LIN {X 0,Y 239.536,Z 764.957,A -85,B 0,C 180,E1 -20171.852,E2 -20171.852} C_VEL
LIN {X 0,Y 237.019,Z 761.771,A -85,B 0,C 180,E1 -20173.722,E2 -20173.722} C_VEL
LIN {X 0,Y 235.633,Z 760.929,A -85,B 0,C 180,E1 -20174.686,E2 -20174.686} C_VEL
LIN {X 0,Y 233.822,Z 758.618,A -85,B 0,C 180,E1 -20176.248,E2 -20176.248} C_VEL
LIN {X 0,Y 232.796,Z 758.036,A -85,B 0,C 180,E1 -20177.061,E2 -20177.061} C_VEL
LIN {X 0,Y 230.567,Z 756.594,A -85,B 0,C 180,E1 -20179.103,E2 -20179.103} C_VEL
LIN {X 0,Y 229.613,Z 755.15,A -85,B 0,C 180,E1 -20180.375,E2 -20180.375} C_VEL
LIN {X 0,Y 230.024,Z 757.239,A -85,B 0,C 180,E1 -20185.325,E2 -20185.325} C_VEL
LIN {X 0,Y 230.532,Z 759.477,A -85,B 0,C 180,E1 -20189.195,E2 -20189.195} C_VEL
LIN {X 0,Y 231.145,Z 762.362,A -85,B 0,C 180,E1 -20193.181,E2 -20193.181} C_VEL
LIN {X 0,Y 232.117,Z 766.675,A -85,B 0,C 180,E1 -20198.073,E2 -20198.073} C_VEL
LIN {X 0,Y 232.844,Z 770.414,A -85,B 0,C 180,E1 -20201.608,E2 -20201.608} C_VEL
LIN {X 0,Y 233.498,Z 773.772,A -85,B 0,C 180,E1 -20204.335,E2 -20204.335} C_VEL
LIN {X 0,Y 235.393,Z 778.757,A -85,B 0,C 180,E1 -20205.95,E2 -20205.95} C_VEL
LIN {X 0,Y 237.78,Z 782.93,A -85,B 0,C 180,E1 -20207.6,E2 -20207.6} C_VEL
LIN {X 0,Y 239.967,Z 789.226,A -85,B 0,C 180,E1 -20209.271,E2 -20209.271} C_VEL
LIN {X 0,Y 241.097,Z 795.425,A -85,B 0,C 180,E1 -20210.543,E2 -20210.543} C_VEL
LIN {X 0,Y 241.775,Z 799.257,A -85,B 0,C 180,E1 -20211.301,E2 -20211.301} C_VEL
LIN {X 0,Y 241.913,Z 804.189,A -85,B 0,C 180,E1 -20212.077,E2 -20212.077} C_VEL
LIN {X 0,Y 241.291,Z 809.401,A -85,B 0,C 180,E1 -20212.744,E2 -20212.744} C_VEL
LIN {X 0,Y 238.925,Z 819.932,A -85,B 0,C 180,E1 -20214.02,E2 -20214.02} C_VEL
LIN {X 0,Y 238.088,Z 824.877,A -85,B 0,C 180,E1 -20214.79,E2 -20214.79} C_VEL
LIN {X 0,Y 238.001,Z 826.424,A -85,B 0,C 180,E1 -20215.084,E2 -20215.084} C_VEL
LIN {X 0,Y 237.022,Z 838.207,A -85,B 0,C 180,E1 -20217.458,E2 -20217.458} C_VEL
LIN {X 0,Y 234.947,Z 849.621,A -85,B 0,C 180,E1 -20219.926,E2 -20219.926} C_VEL
LIN {X 0,Y 231.947,Z 860.19,A -85,B 0,C 180,E1 -20222.479,E2 -20222.479} C_VEL
LIN {X 0,Y 229.183,Z 869.039,A -85,B 0,C 180,E1 -20225.061,E2 -20225.061} C_VEL
LIN {X 0,Y 226.722,Z 875.341,A -85,B 0,C 180,E1 -20227.202,E2 -20227.202} C_VEL
LIN {X 0,Y 223.981,Z 881.748,A -85,B 0,C 180,E1 -20229.808,E2 -20229.808} C_VEL
LIN {X 0,Y 221.954,Z 887.028,A -85,B 0,C 180,E1 -20232.493,E2 -20232.493} C_VEL
LIN {X 0,Y 220.653,Z 891.327,A -85,B 0,C 180,E1 -20235.238,E2 -20235.238} C_VEL
LIN {X 0,Y 219.689,Z 895.654,A -85,B 0,C 180,E1 -20238.933,E2 -20238.933} C_VEL
LIN {X 0,Y 219.717,Z 898.373,A -85,B 0,C 180,E1 -20242.649,E2 -20242.649} C_VEL
LIN {X 0,Y 219.985,Z 899.167,A -85,B 0,C 180,E1 -20244.5,E2 -20244.5} C_VEL
LIN {X 0,Y 220.278,Z 899.554,A -85,B 0,C 180,E1 -20246.341,E2 -20246.341} C_VEL
LIN {X 0,Y 220.658,Z 899.53,A -85,B 0,C 180,E1 -20248.175,E2 -20248.175} C_VEL
LIN {X 0,Y 221.137,Z 899.063,A -85,B 0,C 180,E1 -20250,E2 -20250} C_VEL
LIN {X 0,Y 220.915,Z 898.036,A -85,B 0,C 180,E1 -20251.823,E2 -20251.823} C_VEL
LIN {X 0,Y 220.65,Z 896.554,A -85,B 0,C 180,E1 -20253.652,E2 -20253.652} C_VEL
LIN {X 0,Y 220.44,Z 893.409,A -85,B 0,C 180,E1 -20256.407,E2 -20256.407} C_VEL
LIN {X 0,Y 220.219,Z 889.055,A -85,B 0,C 180,E1 -20259.182,E2 -20259.182} C_VEL
LIN {X 0,Y 220.533,Z 882.364,A -85,B 0,C 180,E1 -20262.422,E2 -20262.422} C_VEL
LIN {X 0,Y 221.328,Z 875.061,A -85,B 0,C 180,E1 -20265.187,E2 -20265.187} C_VEL
LIN {X 0,Y 222.405,Z 867.639,A -85,B 0,C 180,E1 -20267.47,E2 -20267.47} C_VEL
LIN {X 0,Y 223.753,Z 859.408,A -85,B 0,C 180,E1 -20269.56,E2 -20269.56} C_VEL
LIN {X 0,Y 223.898,Z 849.535,A -85,B 0,C 180,E1 -20271.643,E2 -20271.643} C_VEL
LIN {X 0,Y 223.822,Z 838.205,A -85,B 0,C 180,E1 -20273.6,E2 -20273.6} C_VEL
LIN {X 0,Y 223.429,Z 825.557,A -85,B 0,C 180,E1 -20275.376,E2 -20275.376} C_VEL
LIN {X 0,Y 222.909,Z 813.807,A -85,B 0,C 180,E1 -20276.684,E2 -20276.684} C_VEL
LIN {X 0,Y 222.051,Z 799.54,A -85,B 0,C 180,E1 -20277.884,E2 -20277.884} C_VEL
LIN {X 0,Y 221.631,Z 793.027,A -85,B 0,C 180,E1 -20278.33,E2 -20278.33} C_VEL
LIN {X 0,Y 223.268,Z 783.83,A -85,B 0,C 180,E1 -20283.426,E2 -20283.426} C_VEL
LIN {X 0,Y 225.052,Z 776.429,A -85,B 0,C 180,E1 -20287.514,E2 -20287.514} C_VEL
LIN {X 0,Y 225.493,Z 774.103,A -85,B 0,C 180,E1 -20288.814,E2 -20288.814} C_VEL
LIN {X 0,Y 225.149,Z 770.421,A -85,B 0,C 180,E1 -20290.959,E2 -20290.959} C_VEL
LIN {X 0,Y 223.734,Z 763.752,A -85,B 0,C 180,E1 -20295.027,E2 -20295.027} C_VEL
LIN {X 0,Y 222.198,Z 755.968,A -85,B 0,C 180,E1 -20300.027,E2 -20300.027} C_VEL
LIN {X 0,Y 220.923,Z 748.963,A -85,B 0,C 180,E1 -20304.789,E2 -20304.789} C_VEL
LIN {X 0,Y 220.869,Z 748.973,A -85,B 0,C 180,E1 -20309.395,E2 -20309.395} C_VEL
LIN {X 0,Y 220.896,Z 748.965,A -85,B 0,C 180,E1 -20313.55,E2 -20313.55} C_VEL
LIN {X 0,Y 220.867,Z 748.972,A -85,B 0,C 180,E1 -20317.552,E2 -20317.552} C_VEL
LIN {X 0,Y 220.986,Z 748.956,A -85,B 0,C 180,E1 -20322.571,E2 -20322.571} C_VEL
LIN {X 0,Y 221.014,Z 748.952,A -85,B 0,C 180,E1 -20327.139,E2 -20327.139} C_VEL
LIN {X 0,Y 221.207,Z 748.927,A -85,B 0,C 180,E1 -20330.86,E2 -20330.86} C_VEL
LIN {X 0,Y 221.261,Z 748.924,A -85,B 0,C 180,E1 -20332.701,E2 -20332.701} C_VEL
LIN {X 0,Y 221.509,Z 748.89,A -85,B 0,C 180,E1 -20338.182,E2 -20338.182} C_VEL
LIN {X 0,Y 221.51,Z 748.89,A -85,B 0,C 180,E1 -20341.818,E2 -20341.818} C_VEL
LIN {X 0,Y 221.243,Z 748.922,A -85,B 0,C 180,E1 -20347.3,E2 -20347.3} C_VEL
LIN {X 0,Y 221.064,Z 748.95,A -85,B 0,C 180,E1 -20350.997,E2 -20350.997} C_VEL
LIN {X 0,Y 220.992,Z 748.953,A -85,B 0,C 180,E1 -20356.632,E2 -20356.632} C_VEL
LIN {X 0,Y 220.876,Z 748.97,A -85,B 0,C 180,E1 -20360.488,E2 -20360.488} C_VEL
LIN {X 0,Y 220.8,Z 748.976,A -85,B 0,C 180,E1 -20364.443,E2 -20364.443} C_VEL
LIN {X 0,Y 220.801,Z 748.979,A -85,B 0,C 180,E1 -20368.519,E2 -20368.519} C_VEL
LIN {X 0,Y 220.813,Z 748.975,A -85,B 0,C 180,E1 -20372.757,E2 -20372.757} C_VEL
LIN {X 0,Y 220.797,Z 748.98,A -85,B 0,C 180,E1 -20377.274,E2 -20377.274} C_VEL
LIN {X 0,Y 220.747,Z 748.985,A -85,B 0,C 180,E1 -20381.958,E2 -20381.958} C_VEL
LIN {X 0,Y 220.753,Z 748.986,A -85,B 0,C 180,E1 -20385.541,E2 -20385.541} C_VEL
LIN {X 0,Y 220.781,Z 748.979,A -85,B 0,C 180,E1 -20390.458,E2 -20390.458} C_VEL
LIN {X 0,Y 220.826,Z 748.975,A -85,B 0,C 180,E1 -20392.793,E2 -20392.793} C_VEL
LIN {X 0,Y 220.812,Z 748.977,A -85,B 0,C 180,E1 -20397.243,E2 -20397.243} C_VEL
LIN {X 0,Y 220.793,Z 748.978,A -85,B 0,C 180,E1 -20401.48,E2 -20401.48} C_VEL
LIN {X 0,Y 220.806,Z 748.978,A -85,B 0,C 180,E1 -20405.558,E2 -20405.558} C_VEL
LIN {X 0,Y 220.876,Z 748.967,A -85,B 0,C 180,E1 -20409.512,E2 -20409.512} C_VEL
LIN {X 0,Y 220.981,Z 748.957,A -85,B 0,C 180,E1 -20413.368,E2 -20413.368} C_VEL
LIN {X 0,Y 221.064,Z 748.949,A -85,B 0,C 180,E1 -20419.004,E2 -20419.004} C_VEL
LIN {X 0,Y 221.24,Z 748.926,A -85,B 0,C 180,E1 -20422.7,E2 -20422.7} C_VEL
LIN {X 0,Y 221.471,Z 748.895,A -85,B 0,C 180,E1 -20428.182,E2 -20428.182} C_VEL
LIN {X 0,Y 221.471,Z 748.895,A -85,B 0,C 180,E1 -20431.819,E2 -20431.819} C_VEL
LIN {X 0,Y 221.241,Z 748.927,A -85,B 0,C 180,E1 -20437.3,E2 -20437.3} C_VEL
LIN {X 0,Y 221.069,Z 748.946,A -85,B 0,C 180,E1 -20440.997,E2 -20440.997} C_VEL
LIN {X 0,Y 221.02,Z 748.951,A -85,B 0,C 180,E1 -20446.63,E2 -20446.63} C_VEL
LIN {X 0,Y 220.89,Z 748.966,A -85,B 0,C 180,E1 -20450.487,E2 -20450.487} C_VEL
LIN {X 0,Y 220.85,Z 748.973,A -85,B 0,C 180,E1 -20454.437,E2 -20454.437} C_VEL
LIN {X 0,Y 220.807,Z 748.979,A -85,B 0,C 180,E1 -20458.518,E2 -20458.518} C_VEL
LIN {X 0,Y 220.815,Z 748.978,A -85,B 0,C 180,E1 -20462.757,E2 -20462.757} C_VEL
LIN {X 0,Y 220.872,Z 748.986,A -85,B 0,C 180,E1 -20465.851,E2 -20465.851} C_VEL
LIN {X 0,Y 224.644,Z 761.399,A -85,B 0,C 180,E1 -20467.576,E2 -20467.576} C_VEL
LIN {X 0,Y 228.039,Z 773.686,A -85,B 0,C 180,E1 -20469.602,E2 -20469.602} C_VEL
LIN {X 0,Y 228.898,Z 778.294,A -85,B 0,C 180,E1 -20470.437,E2 -20470.437} C_VEL
LIN {X 0,Y 227.328,Z 790.026,A -85,B 0,C 180,E1 -20472.609,E2 -20472.609} C_VEL
LIN {X 0,Y 225.869,Z 799.76,A -85,B 0,C 180,E1 -20474.822,E2 -20474.822} C_VEL
LIN {X 0,Y 224.622,Z 808.015,A -85,B 0,C 180,E1 -20477.116,E2 -20477.116} C_VEL
LIN {X 0,Y 223.342,Z 816.261,A -85,B 0,C 180,E1 -20479.924,E2 -20479.924} C_VEL
LIN {X 0,Y 222.478,Z 822.628,A -85,B 0,C 180,E1 -20482.611,E2 -20482.611} C_VEL
LIN {X 0,Y 221.94,Z 827.949,A -85,B 0,C 180,E1 -20485.42,E2 -20485.42} C_VEL
LIN {X 0,Y 221.554,Z 832.917,A -85,B 0,C 180,E1 -20488.924,E2 -20488.924} C_VEL
LIN {X 0,Y 221.741,Z 836.407,A -85,B 0,C 180,E1 -20492.556,E2 -20492.556} C_VEL
LIN {X 0,Y 222.586,Z 838.266,A -85,B 0,C 180,E1 -20496.3,E2 -20496.3} C_VEL
LIN {X 0,Y 223.975,Z 838.52,A -85,B 0,C 180,E1 -20499.808,E2 -20499.808} C_VEL
LIN {X 0,Y 225.01,Z 837.966,A -85,B 0,C 180,E1 -20501.799,E2 -20501.799} C_VEL
LIN {X 0,Y 226.495,Z 836.725,A -85,B 0,C 180,E1 -20504.137,E2 -20504.137} C_VEL
LIN {X 0,Y 229.235,Z 833.462,A -85,B 0,C 180,E1 -20507.607,E2 -20507.607} C_VEL
LIN {X 0,Y 232.035,Z 829.448,A -85,B 0,C 180,E1 -20510.41,E2 -20510.41} C_VEL
LIN {X 0,Y 235.262,Z 824.148,A -85,B 0,C 180,E1 -20513.137,E2 -20513.137} C_VEL
LIN {X 0,Y 238.765,Z 817.443,A -85,B 0,C 180,E1 -20515.778,E2 -20515.778} C_VEL
LIN {X 0,Y 242.054,Z 810.487,A -85,B 0,C 180,E1 -20517.92,E2 -20517.92} C_VEL
LIN {X 0,Y 245.491,Z 802.175,A -85,B 0,C 180,E1 -20520,E2 -20520} C_VEL
LIN {X 0,Y 245.181,Z 797.388,A -85,B 0,C 180,E1 -20521.642,E2 -20521.642} C_VEL
LIN {X 0,Y 244.015,Z 789.753,A -85,B 0,C 180,E1 -20524.236,E2 -20524.236} C_VEL
LIN {X 0,Y 242.382,Z 784.469,A -85,B 0,C 180,E1 -20526.227,E2 -20526.227} C_VEL
LIN {X 0,Y 238.461,Z 774.826,A -85,B 0,C 180,E1 -20530.185,E2 -20530.185} C_VEL
LIN {X 0,Y 236.378,Z 771.366,A -85,B 0,C 180,E1 -20532.012,E2 -20532.012} C_VEL
LIN {X 0,Y 234.167,Z 768.376,A -85,B 0,C 180,E1 -20533.892,E2 -20533.892} C_VEL
LIN {X 0,Y 229.777,Z 764.406,A -85,B 0,C 180,E1 -20537.81,E2 -20537.81} C_VEL
LIN {X 0,Y 227.615,Z 762.171,A -85,B 0,C 180,E1 -20540.373,E2 -20540.373} C_VEL
LIN {X 0,Y 224.085,Z 761.37,A -85,B 0,C 180,E1 -20546.045,E2 -20546.045} C_VEL
LIN {X 0,Y 223.685,Z 761.148,A -85,B 0,C 180,E1 -20548.118,E2 -20548.118} C_VEL
LIN {X 0,Y 224.259,Z 763.902,A -85,B 0,C 180,E1 -20552.204,E2 -20552.204} C_VEL
LIN {X 0,Y 225.112,Z 767.836,A -85,B 0,C 180,E1 -20556.801,E2 -20556.801} C_VEL
LIN {X 0,Y 228.683,Z 776.557,A -85,B 0,C 180,E1 -20561.863,E2 -20561.863} C_VEL
LIN {X 0,Y 230.667,Z 779.851,A -85,B 0,C 180,E1 -20563.67,E2 -20563.67} C_VEL
LIN {X 0,Y 232.193,Z 784.445,A -85,B 0,C 180,E1 -20565.254,E2 -20565.254} C_VEL
LIN {X 0,Y 234.205,Z 788.172,A -85,B 0,C 180,E1 -20566.81,E2 -20566.81} C_VEL
LIN {X 0,Y 235.872,Z 793.983,A -85,B 0,C 180,E1 -20568.434,E2 -20568.434} C_VEL
LIN {X 0,Y 237.128,Z 803.079,A -85,B 0,C 180,E1 -20570.407,E2 -20570.407} C_VEL
LIN {X 0,Y 238.077,Z 816.236,A -85,B 0,C 180,E1 -20573.062,E2 -20573.062} C_VEL
LIN {X 0,Y 238.001,Z 826.424,A -85,B 0,C 180,E1 -20575.084,E2 -20575.084} C_VEL
LIN {X 0,Y 237.26,Z 831.186,A -85,B 0,C 180,E1 -20575.915,E2 -20575.915} C_VEL
LIN {X 0,Y 235.527,Z 836.054,A -85,B 0,C 180,E1 -20576.636,E2 -20576.636} C_VEL
LIN {X 0,Y 230.95,Z 845.512,A -85,B 0,C 180,E1 -20578.063,E2 -20578.063} C_VEL
LIN {X 0,Y 229.043,Z 849.964,A -85,B 0,C 180,E1 -20578.936,E2 -20578.936} C_VEL
LIN {X 0,Y 228.592,Z 851.381,A -85,B 0,C 180,E1 -20579.268,E2 -20579.268} C_VEL
LIN {X 0,Y 225.114,Z 862.094,A -85,B 0,C 180,E1 -20582.076,E2 -20582.076} C_VEL
LIN {X 0,Y 221.765,Z 871.694,A -85,B 0,C 180,E1 -20585.171,E2 -20585.171} C_VEL
LIN {X 0,Y 218.161,Z 879.44,A -85,B 0,C 180,E1 -20588.255,E2 -20588.255} C_VEL
LIN {X 0,Y 215.692,Z 884.912,A -85,B 0,C 180,E1 -20590.984,E2 -20590.984} C_VEL
LIN {X 0,Y 213.728,Z 890.678,A -85,B 0,C 180,E1 -20594.748,E2 -20594.748} C_VEL
LIN {X 0,Y 212.66,Z 894.779,A -85,B 0,C 180,E1 -20598.563,E2 -20598.563} C_VEL
LIN {X 0,Y 212.673,Z 897.416,A -85,B 0,C 180,E1 -20602.472,E2 -20602.472} C_VEL
LIN {X 0,Y 212.925,Z 898.116,A -85,B 0,C 180,E1 -20604.317,E2 -20604.317} C_VEL
LIN {X 0,Y 213.224,Z 898.43,A -85,B 0,C 180,E1 -20606.22,E2 -20606.22} C_VEL
LIN {X 0,Y 213.649,Z 898.324,A -85,B 0,C 180,E1 -20608.115,E2 -20608.115} C_VEL
LIN {X 0,Y 214.155,Z 897.813,A -85,B 0,C 180,E1 -20610,E2 -20610} C_VEL
LIN {X 0,Y 213.897,Z 896.725,A -85,B 0,C 180,E1 -20611.883,E2 -20611.883} C_VEL
LIN {X 0,Y 213.551,Z 894.183,A -85,B 0,C 180,E1 -20614.719,E2 -20614.719} C_VEL
LIN {X 0,Y 213.289,Z 890.503,A -85,B 0,C 180,E1 -20617.574,E2 -20617.574} C_VEL
LIN {X 0,Y 213.233,Z 885.6,A -85,B 0,C 180,E1 -20620.444,E2 -20620.444} C_VEL
LIN {X 0,Y 213.686,Z 879.386,A -85,B 0,C 180,E1 -20623.31,E2 -20623.31} C_VEL
LIN {X 0,Y 214.678,Z 871.586,A -85,B 0,C 180,E1 -20626.157,E2 -20626.157} C_VEL
LIN {X 0,Y 216.168,Z 861.923,A -85,B 0,C 180,E1 -20628.973,E2 -20628.973} C_VEL
LIN {X 0,Y 216.716,Z 856.865,A -85,B 0,C 180,E1 -20630.204,E2 -20630.204} C_VEL
LIN {X 0,Y 216.786,Z 846.465,A -85,B 0,C 180,E1 -20632.391,E2 -20632.391} C_VEL
LIN {X 0,Y 216.675,Z 834.784,A -85,B 0,C 180,E1 -20634.412,E2 -20634.412} C_VEL
LIN {X 0,Y 216.312,Z 822.268,A -85,B 0,C 180,E1 -20636.145,E2 -20636.145} C_VEL
LIN {X 0,Y 215.674,Z 808.554,A -85,B 0,C 180,E1 -20637.634,E2 -20637.634} C_VEL
LIN {X 0,Y 214.841,Z 794.999,A -85,B 0,C 180,E1 -20638.711,E2 -20638.711} C_VEL
LIN {X 0,Y 214.664,Z 792.094,A -85,B 0,C 180,E1 -20638.898,E2 -20638.898} C_VEL
LIN {X 0,Y 216.195,Z 783.992,A -85,B 0,C 180,E1 -20643.548,E2 -20643.548} C_VEL
LIN {X 0,Y 218.355,Z 775.24,A -85,B 0,C 180,E1 -20648.578,E2 -20648.578} C_VEL
LIN {X 0,Y 218.388,Z 772.741,A -85,B 0,C 180,E1 -20650.063,E2 -20650.063} C_VEL
LIN {X 0,Y 217.183,Z 766.986,A -85,B 0,C 180,E1 -20653.626,E2 -20653.626} C_VEL
LIN {X 0,Y 215.615,Z 759.392,A -85,B 0,C 180,E1 -20658.563,E2 -20658.563} C_VEL
LIN {X 0,Y 214.486,Z 753.23,A -85,B 0,C 180,E1 -20662.79,E2 -20662.79} C_VEL
LIN {X 0,Y 213.855,Z 749.844,A -85,B 0,C 180,E1 -20665.244,E2 -20665.244} C_VEL
LIN {X 0,Y 213.782,Z 749.853,A -85,B 0,C 180,E1 -20670.454,E2 -20670.454} C_VEL
LIN {X 0,Y 213.8,Z 749.85,A -85,B 0,C 180,E1 -20674.702,E2 -20674.702} C_VEL
LIN {X 0,Y 213.805,Z 749.85,A -85,B 0,C 180,E1 -20678.803,E2 -20678.803} C_VEL
LIN {X 0,Y 213.945,Z 749.832,A -85,B 0,C 180,E1 -20682.804,E2 -20682.804} C_VEL
LIN {X 0,Y 213.955,Z 749.833,A -85,B 0,C 180,E1 -20686.707,E2 -20686.707} C_VEL
LIN {X 0,Y 214.144,Z 749.808,A -85,B 0,C 180,E1 -20690.555,E2 -20690.555} C_VEL
LIN {X 0,Y 214.096,Z 749.817,A -85,B 0,C 180,E1 -20694.349,E2 -20694.349} C_VEL
LIN {X 0,Y 214.442,Z 749.77,A -85,B 0,C 180,E1 -20698.122,E2 -20698.122} C_VEL
LIN {X 0,Y 214.544,Z 749.756,A -85,B 0,C 180,E1 -20700,E2 -20700} C_VEL
LIN {X 0,Y 214.443,Z 749.77,A -85,B 0,C 180,E1 -20701.878,E2 -20701.878} C_VEL
LIN {X 0,Y 214.184,Z 749.8,A -85,B 0,C 180,E1 -20707.542,E2 -20707.542} C_VEL
LIN {X 0,Y 213.995,Z 749.828,A -85,B 0,C 180,E1 -20711.365,E2 -20711.365} C_VEL
LIN {X 0,Y 213.91,Z 749.837,A -85,B 0,C 180,E1 -20715.239,E2 -20715.239} C_VEL
LIN {X 0,Y 213.82,Z 749.851,A -85,B 0,C 180,E1 -20719.189,E2 -20719.189} C_VEL
LIN {X 0,Y 213.784,Z 749.855,A -85,B 0,C 180,E1 -20723.235,E2 -20723.235} C_VEL
LIN {X 0,Y 213.786,Z 749.855,A -85,B 0,C 180,E1 -20727.427,E2 -20727.427} C_VEL
LIN {X 0,Y 213.76,Z 749.857,A -85,B 0,C 180,E1 -20731.739,E2 -20731.739} C_VEL
LIN {X 0,Y 213.742,Z 749.859,A -85,B 0,C 180,E1 -20736.289,E2 -20736.289} C_VEL
LIN {X 0,Y 213.697,Z 749.863,A -85,B 0,C 180,E1 -20741.129,E2 -20741.129} C_VEL
LIN {X 0,Y 213.702,Z 749.863,A -85,B 0,C 180,E1 -20743.68,E2 -20743.68} C_VEL
LIN {X 0,Y 213.702,Z 749.865,A -85,B 0,C 180,E1 -20746.346,E2 -20746.346} C_VEL
LIN {X 0,Y 213.702,Z 749.859,A -85,B 0,C 180,E1 -20751.329,E2 -20751.329} C_VEL
LIN {X 0,Y 213.755,Z 749.859,A -85,B 0,C 180,E1 -20756.018,E2 -20756.018} C_VEL
LIN {X 0,Y 213.746,Z 749.858,A -85,B 0,C 180,E1 -20760.449,E2 -20760.449} C_VEL
LIN {X 0,Y 213.742,Z 749.86,A -85,B 0,C 180,E1 -20764.694,E2 -20764.694} C_VEL
LIN {X 0,Y 213.795,Z 749.852,A -85,B 0,C 180,E1 -20768.802,E2 -20768.802} C_VEL
LIN {X 0,Y 213.895,Z 749.842,A -85,B 0,C 180,E1 -20772.8,E2 -20772.8} C_VEL
LIN {X 0,Y 213.937,Z 749.834,A -85,B 0,C 180,E1 -20776.706,E2 -20776.706} C_VEL
LIN {X 0,Y 214.136,Z 749.81,A -85,B 0,C 180,E1 -20780.555,E2 -20780.555} C_VEL
LIN {X 0,Y 214.076,Z 749.816,A -85,B 0,C 180,E1 -20784.348,E2 -20784.348} C_VEL
LIN {X 0,Y 214.407,Z 749.775,A -85,B 0,C 180,E1 -20788.122,E2 -20788.122} C_VEL
LIN {X 0,Y 214.515,Z 749.762,A -85,B 0,C 180,E1 -20790,E2 -20790} C_VEL
LIN {X 0,Y 214.408,Z 749.775,A -85,B 0,C 180,E1 -20791.879,E2 -20791.879} C_VEL
LIN {X 0,Y 214.183,Z 749.806,A -85,B 0,C 180,E1 -20797.542,E2 -20797.542} C_VEL
LIN {X 0,Y 214.001,Z 749.828,A -85,B 0,C 180,E1 -20801.365,E2 -20801.365} C_VEL
LIN {X 0,Y 213.936,Z 749.834,A -85,B 0,C 180,E1 -20805.237,E2 -20805.237} C_VEL
LIN {X 0,Y 213.84,Z 749.847,A -85,B 0,C 180,E1 -20809.188,E2 -20809.188} C_VEL
LIN {X 0,Y 213.806,Z 749.851,A -85,B 0,C 180,E1 -20813.232,E2 -20813.232} C_VEL
LIN {X 0,Y 213.79,Z 749.854,A -85,B 0,C 180,E1 -20817.428,E2 -20817.428} C_VEL
LIN {X 0,Y 213.761,Z 749.859,A -85,B 0,C 180,E1 -20821.739,E2 -20821.739} C_VEL
LIN {X 0,Y 213.794,Z 749.853,A -85,B 0,C 180,E1 -20825.294,E2 -20825.294} C_VEL
LIN {X 0,Y 217.876,Z 763.131,A -85,B 0,C 180,E1 -20827.216,E2 -20827.216} C_VEL
LIN {X 0,Y 220.84,Z 774.127,A -85,B 0,C 180,E1 -20829.093,E2 -20829.093} C_VEL
LIN {X 0,Y 221.943,Z 778.391,A -85,B 0,C 180,E1 -20829.91,E2 -20829.91} C_VEL
LIN {X 0,Y 220.775,Z 788.422,A -85,B 0,C 180,E1 -20831.762,E2 -20831.762} C_VEL
LIN {X 0,Y 219.117,Z 798.981,A -85,B 0,C 180,E1 -20834.138,E2 -20834.138} C_VEL
LIN {X 0,Y 217.708,Z 808.187,A -85,B 0,C 180,E1 -20836.686,E2 -20836.686} C_VEL
LIN {X 0,Y 216.409,Z 816.36,A -85,B 0,C 180,E1 -20839.495,E2 -20839.495} C_VEL
LIN {X 0,Y 215.312,Z 824.119,A -85,B 0,C 180,E1 -20842.853,E2 -20842.853} C_VEL
LIN {X 0,Y 214.73,Z 830.013,A -85,B 0,C 180,E1 -20846.192,E2 -20846.192} C_VEL
LIN {X 0,Y 214.471,Z 834.375,A -85,B 0,C 180,E1 -20849.487,E2 -20849.487} C_VEL
LIN {X 0,Y 214.739,Z 837.379,A -85,B 0,C 180,E1 -20852.729,E2 -20852.729} C_VEL
LIN {X 0,Y 215.445,Z 839.173,A -85,B 0,C 180,E1 -20855.978,E2 -20855.978} C_VEL
LIN {X 0,Y 216.991,Z 839.729,A -85,B 0,C 180,E1 -20859.93,E2 -20859.93} C_VEL
LIN {X 0,Y 219.341,Z 838.449,A -85,B 0,C 180,E1 -20863.997,E2 -20863.997} C_VEL
LIN {X 0,Y 221.803,Z 836.025,A -85,B 0,C 180,E1 -20867.185,E2 -20867.185} C_VEL
LIN {X 0,Y 224.581,Z 832.601,A -85,B 0,C 180,E1 -20870.089,E2 -20870.089} C_VEL
LIN {X 0,Y 227.856,Z 827.892,A -85,B 0,C 180,E1 -20872.913,E2 -20872.913} C_VEL
LIN {X 0,Y 231.435,Z 821.837,A -85,B 0,C 180,E1 -20875.647,E2 -20875.647} C_VEL
LIN {X 0,Y 235.499,Z 814.219,A -85,B 0,C 180,E1 -20878.29,E2 -20878.29} C_VEL
LIN {X 0,Y 239.404,Z 805.721,A -85,B 0,C 180,E1 -20880.588,E2 -20880.588} C_VEL
LIN {X 0,Y 239.801,Z 804.702,A -85,B 0,C 180,E1 -20880.839,E2 -20880.839} C_VEL
LIN {X 0,Y 239.135,Z 795.516,A -85,B 0,C 180,E1 -20884.213,E2 -20884.213} C_VEL
LIN {X 0,Y 238.04,Z 790.733,A -85,B 0,C 180,E1 -20886.083,E2 -20886.083} C_VEL
LIN {X 0,Y 234.694,Z 780.967,A -85,B 0,C 180,E1 -20890.351,E2 -20890.351} C_VEL
LIN {X 0,Y 232.945,Z 777.567,A -85,B 0,C 180,E1 -20892.192,E2 -20892.192} C_VEL
LIN {X 0,Y 231.028,Z 774.762,A -85,B 0,C 180,E1 -20894.085,E2 -20894.085} C_VEL
LIN {X 0,Y 227.118,Z 770.93,A -85,B 0,C 180,E1 -20898.025,E2 -20898.025} C_VEL
LIN {X 0,Y 225.244,Z 768.855,A -85,B 0,C 180,E1 -20900.6,E2 -20900.6} C_VEL
LIN {X 0,Y 222.86,Z 768.528,A -85,B 0,C 180,E1 -20904.202,E2 -20904.202} C_VEL
LIN {X 0,Y 221.879,Z 768.004,A -85,B 0,C 180,E1 -20907.969,E2 -20907.969} C_VEL
LIN {X 0,Y 221.79,Z 771.249,A -85,B 0,C 180,E1 -20912.999,E2 -20912.999} C_VEL
LIN {X 0,Y 223.048,Z 774.544,A -85,B 0,C 180,E1 -20916.471,E2 -20916.471} C_VEL
LIN {X 0,Y 227.449,Z 785.277,A -85,B 0,C 180,E1 -20922.827,E2 -20922.827} C_VEL
LIN {X 0,Y 229.085,Z 790.743,A -85,B 0,C 180,E1 -20924.879,E2 -20924.879} C_VEL
LIN {X 0,Y 230.442,Z 793.382,A -85,B 0,C 180,E1 -20926.03,E2 -20926.03} C_VEL
LIN {X 0,Y 231.488,Z 797.369,A -85,B 0,C 180,E1 -20927.262,E2 -20927.262} C_VEL
LIN {X 0,Y 232.472,Z 807.335,A -85,B 0,C 180,E1 -20929.584,E2 -20929.584} C_VEL
LIN {X 0,Y 232.808,Z 820.657,A -85,B 0,C 180,E1 -20932.471,E2 -20932.471} C_VEL
LIN {X 0,Y 232.104,Z 831.966,A -85,B 0,C 180,E1 -20934.878,E2 -20934.878} C_VEL
LIN {X 0,Y 230.559,Z 842.773,A -85,B 0,C 180,E1 -20937.244,E2 -20937.244} C_VEL
LIN {X 0,Y 228.592,Z 851.381,A -85,B 0,C 180,E1 -20939.268,E2 -20939.268} C_VEL
LIN {X 0,Y 226.806,Z 855.608,A -85,B 0,C 180,E1 -20940.226,E2 -20940.226} C_VEL
LIN {X 0,Y 222.111,Z 862.268,A -85,B 0,C 180,E1 -20941.674,E2 -20941.674} C_VEL
LIN {X 0,Y 218.121,Z 867.224,A -85,B 0,C 180,E1 -20942.914,E2 -20942.914} C_VEL
LIN {X 0,Y 215.772,Z 870.701,A -85,B 0,C 180,E1 -20944.012,E2 -20944.012} C_VEL
LIN {X 0,Y 215.23,Z 871.789,A -85,B 0,C 180,E1 -20944.42,E2 -20944.42} C_VEL
LIN {X 0,Y 211.542,Z 879.206,A -85,B 0,C 180,E1 -20947.538,E2 -20947.538} C_VEL
LIN {X 0,Y 208.958,Z 884.455,A -85,B 0,C 180,E1 -20950.346,E2 -20950.346} C_VEL
LIN {X 0,Y 207.254,Z 888.754,A -85,B 0,C 180,E1 -20953.247,E2 -20953.247} C_VEL
LIN {X 0,Y 206.077,Z 892.144,A -85,B 0,C 180,E1 -20956.188,E2 -20956.188} C_VEL
LIN {X 0,Y 205.481,Z 895.334,A -85,B 0,C 180,E1 -20960.153,E2 -20960.153} C_VEL
LIN {X 0,Y 205.618,Z 896.491,A -85,B 0,C 180,E1 -20962.402,E2 -20962.402} C_VEL
LIN {X 0,Y 205.867,Z 897.031,A -85,B 0,C 180,E1 -20964.121,E2 -20964.121} C_VEL
LIN {X 0,Y 206.634,Z 897.094,A -85,B 0,C 180,E1 -20968.051,E2 -20968.051} C_VEL
LIN {X 0,Y 207.165,Z 896.532,A -85,B 0,C 180,E1 -20970,E2 -20970} C_VEL
LIN {X 0,Y 206.878,Z 895.374,A -85,B 0,C 180,E1 -20971.947,E2 -20971.947} C_VEL
LIN {X 0,Y 206.543,Z 892.724,A -85,B 0,C 180,E1 -20974.88,E2 -20974.88} C_VEL
LIN {X 0,Y 206.251,Z 888.909,A -85,B 0,C 180,E1 -20977.834,E2 -20977.834} C_VEL
LIN {X 0,Y 206.24,Z 883.853,A -85,B 0,C 180,E1 -20980.802,E2 -20980.802} C_VEL
LIN {X 0,Y 206.784,Z 877.45,A -85,B 0,C 180,E1 -20983.763,E2 -20983.763} C_VEL
LIN {X 0,Y 207.853,Z 869.469,A -85,B 0,C 180,E1 -20986.703,E2 -20986.703} C_VEL
LIN {X 0,Y 209.132,Z 861.336,A -85,B 0,C 180,E1 -20989.126,E2 -20989.126} C_VEL
LIN {X 0,Y 209.624,Z 856.536,A -85,B 0,C 180,E1 -20990.357,E2 -20990.357} C_VEL
LIN {X 0,Y 209.738,Z 846.049,A -85,B 0,C 180,E1 -20992.665,E2 -20992.665} C_VEL
LIN {X 0,Y 209.641,Z 834.841,A -85,B 0,C 180,E1 -20994.699,E2 -20994.699} C_VEL
LIN {X 0,Y 209.356,Z 822.205,A -85,B 0,C 180,E1 -20996.545,E2 -20996.545} C_VEL
LIN {X 0,Y 208.74,Z 808.282,A -85,B 0,C 180,E1 -20998.123,E2 -20998.123} C_VEL
LIN {X 0,Y 207.906,Z 794.49,A -85,B 0,C 180,E1 -20999.275,E2 -20999.275} C_VEL
LIN {X 0,Y 207.768,Z 791.111,A -85,B 0,C 180,E1 -20999.527,E2 -20999.527} C_VEL
LIN {X 0,Y 209.528,Z 782.321,A -85,B 0,C 180,E1 -21004.765,E2 -21004.765} C_VEL
LIN {X 0,Y 211.033,Z 776.807,A -85,B 0,C 180,E1 -21008.032,E2 -21008.032} C_VEL
LIN {X 0,Y 211.308,Z 773.421,A -85,B 0,C 180,E1 -21010.096,E2 -21010.096} C_VEL
LIN {X 0,Y 210.098,Z 767.636,A -85,B 0,C 180,E1 -21013.817,E2 -21013.817} C_VEL
LIN {X 0,Y 208.508,Z 760.006,A -85,B 0,C 180,E1 -21018.942,E2 -21018.942} C_VEL
LIN {X 0,Y 207.29,Z 753.421,A -85,B 0,C 180,E1 -21023.608,E2 -21023.608} C_VEL
LIN {X 0,Y 206.79,Z 750.725,A -85,B 0,C 180,E1 -21025.744,E2 -21025.744} C_VEL
LIN {X 0,Y 206.725,Z 750.734,A -85,B 0,C 180,E1 -21029.339,E2 -21029.339} C_VEL
LIN {X 0,Y 206.732,Z 750.73,A -85,B 0,C 180,E1 -21033.772,E2 -21033.772} C_VEL
LIN {X 0,Y 206.741,Z 750.734,A -85,B 0,C 180,E1 -21038.042,E2 -21038.042} C_VEL
LIN {X 0,Y 206.875,Z 750.713,A -85,B 0,C 180,E1 -21042.197,E2 -21042.197} C_VEL
LIN {X 0,Y 206.897,Z 750.715,A -85,B 0,C 180,E1 -21046.245,E2 -21046.245} C_VEL
LIN {X 0,Y 207.101,Z 750.685,A -85,B 0,C 180,E1 -21050.231,E2 -21050.231} C_VEL
LIN {X 0,Y 207.058,Z 750.692,A -85,B 0,C 180,E1 -21054.156,E2 -21054.156} C_VEL
LIN {X 0,Y 207.378,Z 750.65,A -85,B 0,C 180,E1 -21058.058,E2 -21058.058} C_VEL
LIN {X 0,Y 207.509,Z 750.632,A -85,B 0,C 180,E1 -21060,E2 -21060} C_VEL
LIN {X 0,Y 207.379,Z 750.65,A -85,B 0,C 180,E1 -21061.942,E2 -21061.942} C_VEL
LIN {X 0,Y 207.129,Z 750.678,A -85,B 0,C 180,E1 -21067.801,E2 -21067.801} C_VEL
LIN {X 0,Y 206.919,Z 750.709,A -85,B 0,C 180,E1 -21071.759,E2 -21071.759} C_VEL
LIN {X 0,Y 206.844,Z 750.714,A -85,B 0,C 180,E1 -21075.773,E2 -21075.773} C_VEL
LIN {X 0,Y 206.858,Z 750.715,A -85,B 0,C 180,E1 -21077.955,E2 -21077.955} C_VEL
LIN {X 0,Y 206.727,Z 750.733,A -85,B 0,C 180,E1 -21083.378,E2 -21083.378} C_VEL
LIN {X 0,Y 206.688,Z 750.737,A -85,B 0,C 180,E1 -21088.428,E2 -21088.428} C_VEL
LIN {X 0,Y 206.695,Z 750.734,A -85,B 0,C 180,E1 -21092.959,E2 -21092.959} C_VEL
LIN {X 0,Y 206.7,Z 750.734,A -85,B 0,C 180,E1 -21095.311,E2 -21095.311} C_VEL
LIN {X 0,Y 206.646,Z 750.742,A -85,B 0,C 180,E1 -21100.255,E2 -21100.255} C_VEL
LIN {X 0,Y 206.63,Z 750.744,A -85,B 0,C 180,E1 -21104.417,E2 -21104.417} C_VEL
LIN {X 0,Y 206.631,Z 750.744,A -85,B 0,C 180,E1 -21108.442,E2 -21108.442} C_VEL
LIN {X 0,Y 206.666,Z 750.741,A -85,B 0,C 180,E1 -21112.257,E2 -21112.257} C_VEL
LIN {X 0,Y 206.701,Z 750.736,A -85,B 0,C 180,E1 -21114.689,E2 -21114.689} C_VEL
LIN {X 0,Y 206.695,Z 750.732,A -85,B 0,C 180,E1 -21119.334,E2 -21119.334} C_VEL
LIN {X 0,Y 206.681,Z 750.738,A -85,B 0,C 180,E1 -21123.765,E2 -21123.765} C_VEL
LIN {X 0,Y 206.726,Z 750.73,A -85,B 0,C 180,E1 -21128.04,E2 -21128.04} C_VEL
LIN {X 0,Y 206.828,Z 750.72,A -85,B 0,C 180,E1 -21132.193,E2 -21132.193} C_VEL
LIN {X 0,Y 206.878,Z 750.712,A -85,B 0,C 180,E1 -21136.243,E2 -21136.243} C_VEL
LIN {X 0,Y 207.081,Z 750.688,A -85,B 0,C 180,E1 -21140.23,E2 -21140.23} C_VEL
LIN {X 0,Y 207.039,Z 750.692,A -85,B 0,C 180,E1 -21144.155,E2 -21144.155} C_VEL
LIN {X 0,Y 207.347,Z 750.654,A -85,B 0,C 180,E1 -21148.058,E2 -21148.058} C_VEL
LIN {X 0,Y 207.482,Z 750.638,A -85,B 0,C 180,E1 -21150,E2 -21150} C_VEL
LIN {X 0,Y 207.347,Z 750.654,A -85,B 0,C 180,E1 -21151.943,E2 -21151.943} C_VEL
LIN {X 0,Y 207.128,Z 750.684,A -85,B 0,C 180,E1 -21157.801,E2 -21157.801} C_VEL
LIN {X 0,Y 206.926,Z 750.706,A -85,B 0,C 180,E1 -21161.759,E2 -21161.759} C_VEL
LIN {X 0,Y 206.87,Z 750.717,A -85,B 0,C 180,E1 -21165.771,E2 -21165.771} C_VEL
LIN {X 0,Y 206.783,Z 750.726,A -85,B 0,C 180,E1 -21169.869,E2 -21169.869} C_VEL
LIN {X 0,Y 206.741,Z 750.732,A -85,B 0,C 180,E1 -21174.075,E2 -21174.075} C_VEL
LIN {X 0,Y 206.691,Z 750.738,A -85,B 0,C 180,E1 -21178.427,E2 -21178.427} C_VEL
LIN {X 0,Y 206.7,Z 750.737,A -85,B 0,C 180,E1 -21182.958,E2 -21182.958} C_VEL
LIN {X 0,Y 206.734,Z 750.733,A -85,B 0,C 180,E1 -21184.71,E2 -21184.71} C_VEL
LIN {X 0,Y 211.021,Z 764.634,A -85,B 0,C 180,E1 -21186.834,E2 -21186.834} C_VEL
LIN {X 0,Y 214.095,Z 776.208,A -85,B 0,C 180,E1 -21188.889,E2 -21188.889} C_VEL
LIN {X 0,Y 215.02,Z 779.778,A -85,B 0,C 180,E1 -21189.596,E2 -21189.596} C_VEL
LIN {X 0,Y 213.707,Z 790.116,A -85,B 0,C 180,E1 -21191.593,E2 -21191.593} C_VEL
LIN {X 0,Y 211.981,Z 800.853,A -85,B 0,C 180,E1 -21194.126,E2 -21194.126} C_VEL
LIN {X 0,Y 210.622,Z 809.295,A -85,B 0,C 180,E1 -21196.566,E2 -21196.566} C_VEL
LIN {X 0,Y 209.454,Z 816.63,A -85,B 0,C 180,E1 -21199.133,E2 -21199.133} C_VEL
LIN {X 0,Y 208.585,Z 822.632,A -85,B 0,C 180,E1 -21201.67,E2 -21201.67} C_VEL
LIN {X 0,Y 207.904,Z 828.808,A -85,B 0,C 180,E1 -21204.923,E2 -21204.923} C_VEL
LIN {X 0,Y 207.496,Z 833.197,A -85,B 0,C 180,E1 -21207.862,E2 -21207.862} C_VEL
LIN {X 0,Y 207.536,Z 837.373,A -85,B 0,C 180,E1 -21211.699,E2 -21211.699} C_VEL
LIN {X 0,Y 208.305,Z 839.941,A -85,B 0,C 180,E1 -21215.638,E2 -21215.638} C_VEL
LIN {X 0,Y 209.823,Z 840.937,A -85,B 0,C 180,E1 -21219.696,E2 -21219.696} C_VEL
LIN {X 0,Y 211.393,Z 840.564,A -85,B 0,C 180,E1 -21222.589,E2 -21222.589} C_VEL
LIN {X 0,Y 212.758,Z 839.705,A -85,B 0,C 180,E1 -21224.677,E2 -21224.677} C_VEL
LIN {X 0,Y 215.503,Z 837.264,A -85,B 0,C 180,E1 -21228.062,E2 -21228.062} C_VEL
LIN {X 0,Y 218.145,Z 834.253,A -85,B 0,C 180,E1 -21230.73,E2 -21230.73} C_VEL
LIN {X 0,Y 221.615,Z 829.701,A -85,B 0,C 180,E1 -21233.627,E2 -21233.627} C_VEL
LIN {X 0,Y 225.895,Z 823.063,A -85,B 0,C 180,E1 -21236.756,E2 -21236.756} C_VEL
LIN {X 0,Y 229.661,Z 816.459,A -85,B 0,C 180,E1 -21239.123,E2 -21239.123} C_VEL
LIN {X 0,Y 233.474,Z 808.832,A -85,B 0,C 180,E1 -21241.304,E2 -21241.304} C_VEL
LIN {X 0,Y 234.073,Z 807.308,A -85,B 0,C 180,E1 -21241.72,E2 -21241.72} C_VEL
LIN {X 0,Y 233.826,Z 799.697,A -85,B 0,C 180,E1 -21244.741,E2 -21244.741} C_VEL
LIN {X 0,Y 233.282,Z 796.233,A -85,B 0,C 180,E1 -21246.18,E2 -21246.18} C_VEL
LIN {X 0,Y 230.676,Z 786.922,A -85,B 0,C 180,E1 -21250.533,E2 -21250.533} C_VEL
LIN {X 0,Y 229.232,Z 783.596,A -85,B 0,C 180,E1 -21252.393,E2 -21252.393} C_VEL
LIN {X 0,Y 227.608,Z 780.928,A -85,B 0,C 180,E1 -21254.301,E2 -21254.301} C_VEL
LIN {X 0,Y 224.17,Z 777.296,A -85,B 0,C 180,E1 -21258.271,E2 -21258.271} C_VEL
LIN {X 0,Y 222.818,Z 775.882,A -85,B 0,C 180,E1 -21260.301,E2 -21260.301} C_VEL
LIN {X 0,Y 220.422,Z 775.163,A -85,B 0,C 180,E1 -21264.487,E2 -21264.487} C_VEL
LIN {X 0,Y 219.915,Z 774.846,A -85,B 0,C 180,E1 -21266.578,E2 -21266.578} C_VEL
LIN {X 0,Y 219.541,Z 775.22,A -85,B 0,C 180,E1 -21268.697,E2 -21268.697} C_VEL
LIN {X 0,Y 219.839,Z 778.775,A -85,B 0,C 180,E1 -21273.778,E2 -21273.778} C_VEL
LIN {X 0,Y 220.229,Z 779.903,A -85,B 0,C 180,E1 -21275.059,E2 -21275.059} C_VEL
LIN {X 0,Y 221.092,Z 783.123,A -85,B 0,C 180,E1 -21277.373,E2 -21277.373} C_VEL
LIN {X 0,Y 224.233,Z 791.557,A -85,B 0,C 180,E1 -21282.342,E2 -21282.342} C_VEL
LIN {X 0,Y 225.47,Z 796.207,A -85,B 0,C 180,E1 -21284.199,E2 -21284.199} C_VEL
LIN {X 0,Y 226.667,Z 799.185,A -85,B 0,C 180,E1 -21285.491,E2 -21285.491} C_VEL
LIN {X 0,Y 227.438,Z 803.817,A -85,B 0,C 180,E1 -21286.889,E2 -21286.889} C_VEL
LIN {X 0,Y 227.719,Z 815.092,A -85,B 0,C 180,E1 -21289.6,E2 -21289.6} C_VEL
LIN {X 0,Y 227.278,Z 825.824,A -85,B 0,C 180,E1 -21292.078,E2 -21292.078} C_VEL
LIN {X 0,Y 226.03,Z 836.738,A -85,B 0,C 180,E1 -21294.571,E2 -21294.571} C_VEL
LIN {X 0,Y 223.733,Z 847.668,A -85,B 0,C 180,E1 -21297.189,E2 -21297.189} C_VEL
LIN {X 0,Y 221.137,Z 856.324,A -85,B 0,C 180,E1 -21299.436,E2 -21299.436} C_VEL
LIN {X 0,Y 217.795,Z 865.252,A -85,B 0,C 180,E1 -21302.102,E2 -21302.102} C_VEL
LIN {X 0,Y 215.23,Z 871.789,A -85,B 0,C 180,E1 -21304.42,E2 -21304.42} C_VEL
LIN {X 0,Y 213.149,Z 875.035,A -85,B 0,C 180,E1 -21305.629,E2 -21305.629} C_VEL
LIN {X 0,Y 207.959,Z 879.818,A -85,B 0,C 180,E1 -21307.542,E2 -21307.542} C_VEL
LIN {X 0,Y 202.972,Z 883.926,A -85,B 0,C 180,E1 -21309.636,E2 -21309.636} C_VEL
LIN {X 0,Y 201.255,Z 886.094,A -85,B 0,C 180,E1 -21311.099,E2 -21311.099} C_VEL
LIN {X 0,Y 199.509,Z 890.405,A -85,B 0,C 180,E1 -21314.68,E2 -21314.68} C_VEL
LIN {X 0,Y 198.65,Z 893.078,A -85,B 0,C 180,E1 -21317.744,E2 -21317.744} C_VEL
LIN {X 0,Y 198.5,Z 895.337,A -85,B 0,C 180,E1 -21321.858,E2 -21321.858} C_VEL
LIN {X 0,Y 198.809,Z 895.911,A -85,B 0,C 180,E1 -21323.912,E2 -21323.912} C_VEL
LIN {X 0,Y 199.613,Z 895.871,A -85,B 0,C 180,E1 -21327.982,E2 -21327.982} C_VEL
LIN {X 0,Y 200.17,Z 895.24,A -85,B 0,C 180,E1 -21330,E2 -21330} C_VEL
LIN {X 0,Y 199.886,Z 893.96,A -85,B 0,C 180,E1 -21332.015,E2 -21332.015} C_VEL
LIN {X 0,Y 199.529,Z 891.171,A -85,B 0,C 180,E1 -21335.052,E2 -21335.052} C_VEL
LIN {X 0,Y 199.241,Z 887.197,A -85,B 0,C 180,E1 -21338.111,E2 -21338.111} C_VEL
LIN {X 0,Y 199.359,Z 880.992,A -85,B 0,C 180,E1 -21341.695,E2 -21341.695} C_VEL
LIN {X 0,Y 200.013,Z 874.169,A -85,B 0,C 180,E1 -21344.759,E2 -21344.759} C_VEL
LIN {X 0,Y 201.252,Z 865.625,A -85,B 0,C 180,E1 -21347.792,E2 -21347.792} C_VEL
LIN {X 0,Y 202.412,Z 858.826,A -85,B 0,C 180,E1 -21349.787,E2 -21349.787} C_VEL
LIN {X 0,Y 202.644,Z 849.14,A -85,B 0,C 180,E1 -21352.158,E2 -21352.158} C_VEL
LIN {X 0,Y 202.705,Z 838.512,A -85,B 0,C 180,E1 -21354.313,E2 -21354.313} C_VEL
LIN {X 0,Y 202.446,Z 826.841,A -85,B 0,C 180,E1 -21356.259,E2 -21356.259} C_VEL
LIN {X 0,Y 202.028,Z 813.547,A -85,B 0,C 180,E1 -21358.01,E2 -21358.01} C_VEL
LIN {X 0,Y 201.367,Z 800.215,A -85,B 0,C 180,E1 -21359.366,E2 -21359.366} C_VEL
LIN {X 0,Y 200.849,Z 790.106,A -85,B 0,C 180,E1 -21360.177,E2 -21360.177} C_VEL
LIN {X 0,Y 202.948,Z 780.602,A -85,B 0,C 180,E1 -21366.065,E2 -21366.065} C_VEL
LIN {X 0,Y 203.998,Z 776.935,A -85,B 0,C 180,E1 -21368.325,E2 -21368.325} C_VEL
LIN {X 0,Y 204.262,Z 775.115,A -85,B 0,C 180,E1 -21369.471,E2 -21369.471} C_VEL
LIN {X 0,Y 203.59,Z 770.998,A -85,B 0,C 180,E1 -21372.155,E2 -21372.155} C_VEL
LIN {X 0,Y 202.078,Z 764.016,A -85,B 0,C 180,E1 -21376.916,E2 -21376.916} C_VEL
LIN {X 0,Y 200.688,Z 756.654,A -85,B 0,C 180,E1 -21382.205,E2 -21382.205} C_VEL
LIN {X 0,Y 199.724,Z 751.606,A -85,B 0,C 180,E1 -21386.132,E2 -21386.132} C_VEL
LIN {X 0,Y 199.676,Z 751.61,A -85,B 0,C 180,E1 -21390.478,E2 -21390.478} C_VEL
LIN {X 0,Y 199.666,Z 751.61,A -85,B 0,C 180,E1 -21395.015,E2 -21395.015} C_VEL
LIN {X 0,Y 199.692,Z 751.608,A -85,B 0,C 180,E1 -21399.394,E2 -21399.394} C_VEL
LIN {X 0,Y 199.807,Z 751.593,A -85,B 0,C 180,E1 -21403.657,E2 -21403.657} C_VEL
LIN {X 0,Y 199.881,Z 751.586,A -85,B 0,C 180,E1 -21407.821,E2 -21407.821} C_VEL
LIN {X 0,Y 200.091,Z 751.557,A -85,B 0,C 180,E1 -21411.924,E2 -21411.924} C_VEL
LIN {X 0,Y 200.318,Z 751.529,A -85,B 0,C 180,E1 -21417.99,E2 -21417.99} C_VEL
LIN {X 0,Y 200.474,Z 751.508,A -85,B 0,C 180,E1 -21420,E2 -21420} C_VEL
LIN {X 0,Y 200.018,Z 751.568,A -85,B 0,C 180,E1 -21424.03,E2 -21424.03} C_VEL
LIN {X 0,Y 200.077,Z 751.556,A -85,B 0,C 180,E1 -21428.077,E2 -21428.077} C_VEL
LIN {X 0,Y 199.868,Z 751.587,A -85,B 0,C 180,E1 -21432.18,E2 -21432.18} C_VEL
LIN {X 0,Y 199.788,Z 751.593,A -85,B 0,C 180,E1 -21436.345,E2 -21436.345} C_VEL
LIN {X 0,Y 199.671,Z 751.612,A -85,B 0,C 180,E1 -21440.609,E2 -21440.609} C_VEL
LIN {X 0,Y 199.626,Z 751.615,A -85,B 0,C 180,E1 -21444.991,E2 -21444.991} C_VEL
LIN {X 0,Y 199.609,Z 751.622,A -85,B 0,C 180,E1 -21449.533,E2 -21449.533} C_VEL
LIN {X 0,Y 199.666,Z 751.609,A -85,B 0,C 180,E1 -21452.353,E2 -21452.353} C_VEL
LIN {X 0,Y 199.616,Z 751.618,A -85,B 0,C 180,E1 -21456.765,E2 -21456.765} C_VEL
LIN {X 0,Y 199.594,Z 751.622,A -85,B 0,C 180,E1 -21459.332,E2 -21459.332} C_VEL
LIN {X 0,Y 199.566,Z 751.622,A -85,B 0,C 180,E1 -21462.307,E2 -21462.307} C_VEL
LIN {X 0,Y 199.576,Z 751.623,A -85,B 0,C 180,E1 -21465.228,E2 -21465.228} C_VEL
LIN {X 0,Y 199.57,Z 751.626,A -85,B 0,C 180,E1 -21468.003,E2 -21468.003} C_VEL
LIN {X 0,Y 199.597,Z 751.616,A -85,B 0,C 180,E1 -21470.773,E2 -21470.773} C_VEL
LIN {X 0,Y 199.612,Z 751.62,A -85,B 0,C 180,E1 -21475.713,E2 -21475.713} C_VEL
LIN {X 0,Y 199.687,Z 751.611,A -85,B 0,C 180,E1 -21478.135,E2 -21478.135} C_VEL
LIN {X 0,Y 199.627,Z 751.618,A -85,B 0,C 180,E1 -21482.763,E2 -21482.763} C_VEL
LIN {X 0,Y 199.677,Z 751.608,A -85,B 0,C 180,E1 -21487.222,E2 -21487.222} C_VEL
LIN {X 0,Y 199.752,Z 751.601,A -85,B 0,C 180,E1 -21491.799,E2 -21491.799} C_VEL
LIN {X 0,Y 199.816,Z 751.591,A -85,B 0,C 180,E1 -21495.747,E2 -21495.747} C_VEL
LIN {X 0,Y 200.025,Z 751.567,A -85,B 0,C 180,E1 -21499.882,E2 -21499.882} C_VEL
LIN {X 0,Y 200.003,Z 751.568,A -85,B 0,C 180,E1 -21503.949,E2 -21503.949} C_VEL
LIN {X 0,Y 200.289,Z 751.533,A -85,B 0,C 180,E1 -21507.989,E2 -21507.989} C_VEL
LIN {X 0,Y 200.45,Z 751.514,A -85,B 0,C 180,E1 -21510,E2 -21510} C_VEL
LIN {X 0,Y 199.993,Z 751.567,A -85,B 0,C 180,E1 -21514.03,E2 -21514.03} C_VEL
LIN {X 0,Y 200.076,Z 751.561,A -85,B 0,C 180,E1 -21518.077,E2 -21518.077} C_VEL
LIN {X 0,Y 199.876,Z 751.582,A -85,B 0,C 180,E1 -21522.18,E2 -21522.18} C_VEL
LIN {X 0,Y 199.808,Z 751.594,A -85,B 0,C 180,E1 -21526.344,E2 -21526.344} C_VEL
LIN {X 0,Y 199.694,Z 751.606,A -85,B 0,C 180,E1 -21530.606,E2 -21530.606} C_VEL
LIN {X 0,Y 199.654,Z 751.613,A -85,B 0,C 180,E1 -21534.987,E2 -21534.987} C_VEL
LIN {X 0,Y 199.611,Z 751.62,A -85,B 0,C 180,E1 -21539.533,E2 -21539.533} C_VEL
LIN {X 0,Y 199.684,Z 751.613,A -85,B 0,C 180,E1 -21543.98,E2 -21543.98} C_VEL
LIN {X 0,Y 199.676,Z 751.614,A -85,B 0,C 180,E1 -21544.128,E2 -21544.128} C_VEL
LIN {X 0,Y 203.764,Z 764.826,A -85,B 0,C 180,E1 -21546.204,E2 -21546.204} C_VEL
LIN {X 0,Y 206.586,Z 775.295,A -85,B 0,C 180,E1 -21548.101,E2 -21548.101} C_VEL
LIN {X 0,Y 208.101,Z 781.195,A -85,B 0,C 180,E1 -21549.298,E2 -21549.298} C_VEL
LIN {X 0,Y 206.532,Z 792.246,A -85,B 0,C 180,E1 -21551.528,E2 -21551.528} C_VEL
LIN {X 0,Y 204.755,Z 803.128,A -85,B 0,C 180,E1 -21554.232,E2 -21554.232} C_VEL
LIN {X 0,Y 203.276,Z 812.063,A -85,B 0,C 180,E1 -21557.007,E2 -21557.007} C_VEL
LIN {X 0,Y 202.022,Z 819.775,A -85,B 0,C 180,E1 -21559.938,E2 -21559.938} C_VEL
LIN {X 0,Y 201.139,Z 826.147,A -85,B 0,C 180,E1 -21562.935,E2 -21562.935} C_VEL
LIN {X 0,Y 200.637,Z 831.223,A -85,B 0,C 180,E1 -21565.912,E2 -21565.912} C_VEL
LIN {X 0,Y 200.377,Z 835.853,A -85,B 0,C 180,E1 -21569.431,E2 -21569.431} C_VEL
LIN {X 0,Y 200.647,Z 839.117,A -85,B 0,C 180,E1 -21572.912,E2 -21572.912} C_VEL
LIN {X 0,Y 201.165,Z 840.673,A -85,B 0,C 180,E1 -21575.279,E2 -21575.279} C_VEL
LIN {X 0,Y 201.847,Z 841.59,A -85,B 0,C 180,E1 -21577.48,E2 -21577.48} C_VEL
LIN {X 0,Y 202.795,Z 842.052,A -85,B 0,C 180,E1 -21579.723,E2 -21579.723} C_VEL
LIN {X 0,Y 203.943,Z 842.042,A -85,B 0,C 180,E1 -21581.932,E2 -21581.932} C_VEL
LIN {X 0,Y 205.273,Z 841.519,A -85,B 0,C 180,E1 -21584.103,E2 -21584.103} C_VEL
LIN {X 0,Y 206.875,Z 840.551,A -85,B 0,C 180,E1 -21586.243,E2 -21586.243} C_VEL
LIN {X 0,Y 208.642,Z 839.071,A -85,B 0,C 180,E1 -21588.34,E2 -21588.34} C_VEL
LIN {X 0,Y 211.755,Z 835.921,A -85,B 0,C 180,E1 -21591.411,E2 -21591.411} C_VEL
LIN {X 0,Y 215.399,Z 831.566,A -85,B 0,C 180,E1 -21594.382,E2 -21594.382} C_VEL
LIN {X 0,Y 219.524,Z 825.76,A -85,B 0,C 180,E1 -21597.328,E2 -21597.328} C_VEL
LIN {X 0,Y 223.867,Z 818.74,A -85,B 0,C 180,E1 -21600,E2 -21600} C_VEL
LIN {X 0,Y 228.258,Z 810.643,A -85,B 0,C 180,E1 -21602.426,E2 -21602.426} C_VEL
LIN {X 0,Y 228.505,Z 803.789,A -85,B 0,C 180,E1 -21605.294,E2 -21605.294} C_VEL
LIN {X 0,Y 228.027,Z 799.954,A -85,B 0,C 180,E1 -21607.081,E2 -21607.081} C_VEL
LIN {X 0,Y 226.398,Z 792.698,A -85,B 0,C 180,E1 -21610.734,E2 -21610.734} C_VEL
LIN {X 0,Y 225.291,Z 789.464,A -85,B 0,C 180,E1 -21612.613,E2 -21612.613} C_VEL
LIN {X 0,Y 223.916,Z 786.92,A -85,B 0,C 180,E1 -21614.542,E2 -21614.542} C_VEL
LIN {X 0,Y 220.93,Z 783.532,A -85,B 0,C 180,E1 -21618.549,E2 -21618.549} C_VEL
LIN {X 0,Y 219.745,Z 782.308,A -85,B 0,C 180,E1 -21620.598,E2 -21620.598} C_VEL
LIN {X 0,Y 217.304,Z 781.542,A -85,B 0,C 180,E1 -21626.922,E2 -21626.922} C_VEL
LIN {X 0,Y 217.011,Z 782.176,A -85,B 0,C 180,E1 -21629.064,E2 -21629.064} C_VEL
LIN {X 0,Y 217.462,Z 785.903,A -85,B 0,C 180,E1 -21634.198,E2 -21634.198} C_VEL
LIN {X 0,Y 218.031,Z 788.434,A -85,B 0,C 180,E1 -21636.307,E2 -21636.307} C_VEL
LIN {X 0,Y 220.512,Z 796.761,A -85,B 0,C 180,E1 -21641.44,E2 -21641.44} C_VEL
LIN {X 0,Y 222.783,Z 805.545,A -85,B 0,C 180,E1 -21645.222,E2 -21645.222} C_VEL
LIN {X 0,Y 223.035,Z 810.979,A -85,B 0,C 180,E1 -21646.747,E2 -21646.747} C_VEL
LIN {X 0,Y 222.372,Z 824.123,A -85,B 0,C 180,E1 -21650.051,E2 -21650.051} C_VEL
LIN {X 0,Y 220.889,Z 835.337,A -85,B 0,C 180,E1 -21652.805,E2 -21652.805} C_VEL
LIN {X 0,Y 218.827,Z 845.095,A -85,B 0,C 180,E1 -21655.244,E2 -21655.244} C_VEL
LIN {X 0,Y 216.016,Z 854.407,A -85,B 0,C 180,E1 -21657.768,E2 -21657.768} C_VEL
LIN {X 0,Y 212.061,Z 864.201,A -85,B 0,C 180,E1 -21660.736,E2 -21660.736} C_VEL
LIN {X 0,Y 208.337,Z 872.824,A -85,B 0,C 180,E1 -21663.989,E2 -21663.989} C_VEL
LIN {X 0,Y 203.999,Z 880.747,A -85,B 0,C 180,E1 -21667.73,E2 -21667.73} C_VEL
LIN {X 0,Y 201.255,Z 886.094,A -85,B 0,C 180,E1 -21671.099,E2 -21671.099} C_VEL
LIN {X 0,Y 199.751,Z 888.134,A -85,B 0,C 180,E1 -21672.628,E2 -21672.628} C_VEL
LIN {X 0,Y 195.797,Z 890.743,A -85,B 0,C 180,E1 -21675.15,E2 -21675.15} C_VEL
LIN {X 0,Y 192.246,Z 892.638,A -85,B 0,C 180,E1 -21677.827,E2 -21677.827} C_VEL
LIN {X 0,Y 191.406,Z 893.469,A -85,B 0,C 180,E1 -21679.556,E2 -21679.556} C_VEL
LIN {X 0,Y 191.749,Z 894.79,A -85,B 0,C 180,E1 -21683.687,E2 -21683.687} C_VEL
LIN {X 0,Y 192.08,Z 894.9,A -85,B 0,C 180,E1 -21685.803,E2 -21685.803} C_VEL
LIN {X 0,Y 192.588,Z 894.606,A -85,B 0,C 180,E1 -21687.908,E2 -21687.908} C_VEL
LIN {X 0,Y 193.194,Z 893.887,A -85,B 0,C 180,E1 -21690,E2 -21690} C_VEL
LIN {X 0,Y 192.89,Z 892.547,A -85,B 0,C 180,E1 -21692.088,E2 -21692.088} C_VEL
LIN {X 0,Y 192.511,Z 889.61,A -85,B 0,C 180,E1 -21695.236,E2 -21695.236} C_VEL
LIN {X 0,Y 192.211,Z 885.476,A -85,B 0,C 180,E1 -21698.41,E2 -21698.41} C_VEL
LIN {X 0,Y 192.342,Z 880.1,A -85,B 0,C 180,E1 -21701.593,E2 -21701.593} C_VEL
LIN {X 0,Y 192.982,Z 873.328,A -85,B 0,C 180,E1 -21704.769,E2 -21704.769} C_VEL
LIN {X 0,Y 194.21,Z 864.834,A -85,B 0,C 180,E1 -21707.914,E2 -21707.914} C_VEL
LIN {X 0,Y 195.431,Z 857.047,A -85,B 0,C 180,E1 -21710.265,E2 -21710.265} C_VEL
LIN {X 0,Y 195.585,Z 847.228,A -85,B 0,C 180,E1 -21712.723,E2 -21712.723} C_VEL
LIN {X 0,Y 195.572,Z 836.37,A -85,B 0,C 180,E1 -21714.976,E2 -21714.976} C_VEL
LIN {X 0,Y 195.391,Z 823.769,A -85,B 0,C 180,E1 -21717.081,E2 -21717.081} C_VEL
LIN {X 0,Y 194.936,Z 810.177,A -85,B 0,C 180,E1 -21718.883,E2 -21718.883} C_VEL
LIN {X 0,Y 194.278,Z 796.122,A -85,B 0,C 180,E1 -21720.266,E2 -21720.266} C_VEL
LIN {X 0,Y 193.912,Z 789.229,A -85,B 0,C 180,E1 -21720.793,E2 -21720.793} C_VEL
LIN {X 0,Y 196.431,Z 778.857,A -85,B 0,C 180,E1 -21727.462,E2 -21727.462} C_VEL
LIN {X 0,Y 197.052,Z 776.525,A -85,B 0,C 180,E1 -21728.954,E2 -21728.954} C_VEL
LIN {X 0,Y 197.044,Z 773.978,A -85,B 0,C 180,E1 -21730.638,E2 -21730.638} C_VEL
LIN {X 0,Y 195.328,Z 766.26,A -85,B 0,C 180,E1 -21736.022,E2 -21736.022} C_VEL
LIN {X 0,Y 194.08,Z 759.912,A -85,B 0,C 180,E1 -21740.676,E2 -21740.676} C_VEL
LIN {X 0,Y 192.894,Z 753.522,A -85,B 0,C 180,E1 -21745.616,E2 -21745.616} C_VEL
LIN {X 0,Y 192.689,Z 752.481,A -85,B 0,C 180,E1 -21746.519,E2 -21746.519} C_VEL
LIN {X 0,Y 192.666,Z 752.485,A -85,B 0,C 180,E1 -21751.692,E2 -21751.692} C_VEL
LIN {X 0,Y 192.686,Z 752.483,A -85,B 0,C 180,E1 -21756.346,E2 -21756.346} C_VEL
LIN {X 0,Y 192.733,Z 752.472,A -85,B 0,C 180,E1 -21761.458,E2 -21761.458} C_VEL
LIN {X 0,Y 192.766,Z 752.471,A -85,B 0,C 180,E1 -21765.214,E2 -21765.214} C_VEL
LIN {X 0,Y 192.946,Z 752.446,A -85,B 0,C 180,E1 -21769.567,E2 -21769.567} C_VEL
LIN {X 0,Y 193.038,Z 752.435,A -85,B 0,C 180,E1 -21771.626,E2 -21771.626} C_VEL
LIN {X 0,Y 193.259,Z 752.408,A -85,B 0,C 180,E1 -21777.916,E2 -21777.916} C_VEL
LIN {X 0,Y 193.439,Z 752.384,A -85,B 0,C 180,E1 -21780,E2 -21780} C_VEL
LIN {X 0,Y 192.964,Z 752.447,A -85,B 0,C 180,E1 -21784.178,E2 -21784.178} C_VEL
LIN {X 0,Y 193.027,Z 752.435,A -85,B 0,C 180,E1 -21788.374,E2 -21788.374} C_VEL
LIN {X 0,Y 192.795,Z 752.469,A -85,B 0,C 180,E1 -21792.634,E2 -21792.634} C_VEL
LIN {X 0,Y 192.748,Z 752.471,A -85,B 0,C 180,E1 -21796.96,E2 -21796.96} C_VEL
LIN {X 0,Y 192.595,Z 752.495,A -85,B 0,C 180,E1 -21801.402,E2 -21801.402} C_VEL
LIN {X 0,Y 192.621,Z 752.486,A -85,B 0,C 180,E1 -21804.195,E2 -21804.195} C_VEL
LIN {X 0,Y 192.602,Z 752.492,A -85,B 0,C 180,E1 -21808.865,E2 -21808.865} C_VEL
LIN {X 0,Y 192.595,Z 752.491,A -85,B 0,C 180,E1 -21813.187,E2 -21813.187} C_VEL
LIN {X 0,Y 192.541,Z 752.5,A -85,B 0,C 180,E1 -21818.355,E2 -21818.355} C_VEL
LIN {X 0,Y 192.485,Z 752.503,A -85,B 0,C 180,E1 -21823.093,E2 -21823.093} C_VEL
LIN {X 0,Y 192.485,Z 752.506,A -85,B 0,C 180,E1 -21826.907,E2 -21826.907} C_VEL
LIN {X 0,Y 192.541,Z 752.496,A -85,B 0,C 180,E1 -21831.646,E2 -21831.646} C_VEL
LIN {X 0,Y 192.596,Z 752.492,A -85,B 0,C 180,E1 -21836.814,E2 -21836.814} C_VEL
LIN {X 0,Y 192.612,Z 752.489,A -85,B 0,C 180,E1 -21841.684,E2 -21841.684} C_VEL
LIN {X 0,Y 192.659,Z 752.487,A -85,B 0,C 180,E1 -21846.343,E2 -21846.343} C_VEL
LIN {X 0,Y 192.7,Z 752.479,A -85,B 0,C 180,E1 -21851.489,E2 -21851.489} C_VEL
LIN {X 0,Y 192.742,Z 752.473,A -85,B 0,C 180,E1 -21855.212,E2 -21855.212} C_VEL
LIN {X 0,Y 192.948,Z 752.449,A -85,B 0,C 180,E1 -21859.567,E2 -21859.567} C_VEL
LIN {X 0,Y 192.967,Z 752.445,A -85,B 0,C 180,E1 -21863.727,E2 -21863.727} C_VEL
LIN {X 0,Y 193.233,Z 752.412,A -85,B 0,C 180,E1 -21867.916,E2 -21867.916} C_VEL
LIN {X 0,Y 193.416,Z 752.391,A -85,B 0,C 180,E1 -21870,E2 -21870} C_VEL
LIN {X 0,Y 192.94,Z 752.445,A -85,B 0,C 180,E1 -21874.178,E2 -21874.178} C_VEL
LIN {X 0,Y 193.027,Z 752.439,A -85,B 0,C 180,E1 -21878.374,E2 -21878.374} C_VEL
LIN {X 0,Y 192.804,Z 752.463,A -85,B 0,C 180,E1 -21882.634,E2 -21882.634} C_VEL
LIN {X 0,Y 192.761,Z 752.472,A -85,B 0,C 180,E1 -21886.959,E2 -21886.959} C_VEL
LIN {X 0,Y 192.623,Z 752.488,A -85,B 0,C 180,E1 -21891.399,E2 -21891.399} C_VEL
LIN {X 0,Y 192.642,Z 752.488,A -85,B 0,C 180,E1 -21894.208,E2 -21894.208} C_VEL
LIN {X 0,Y 192.604,Z 752.492,A -85,B 0,C 180,E1 -21898.866,E2 -21898.866} C_VEL
LIN {X 0,Y 192.66,Z 752.572,A -85,B 0,C 180,E1 -21903.565,E2 -21903.565} C_VEL
LIN {X 0,Y 196.476,Z 765.02,A -85,B 0,C 180,E1 -21905.54,E2 -21905.54} C_VEL
LIN {X 0,Y 199.235,Z 774.948,A -85,B 0,C 180,E1 -21907.377,E2 -21907.377} C_VEL
LIN {X 0,Y 201.157,Z 782.56,A -85,B 0,C 180,E1 -21908.968,E2 -21908.968} C_VEL
LIN {X 0,Y 199.357,Z 794.491,A -85,B 0,C 180,E1 -21911.484,E2 -21911.484} C_VEL
LIN {X 0,Y 197.745,Z 804.038,A -85,B 0,C 180,E1 -21913.97,E2 -21913.97} C_VEL
LIN {X 0,Y 196.088,Z 813.638,A -85,B 0,C 180,E1 -21917.079,E2 -21917.079} C_VEL
LIN {X 0,Y 194.846,Z 821.41,A -85,B 0,C 180,E1 -21920.19,E2 -21920.19} C_VEL
LIN {X 0,Y 193.944,Z 828.331,A -85,B 0,C 180,E1 -21923.675,E2 -21923.675} C_VEL
LIN {X 0,Y 193.45,Z 833.496,A -85,B 0,C 180,E1 -21926.978,E2 -21926.978} C_VEL
LIN {X 0,Y 193.335,Z 837.972,A -85,B 0,C 180,E1 -21930.743,E2 -21930.743} C_VEL
LIN {X 0,Y 194.004,Z 841.274,A -85,B 0,C 180,E1 -21934.912,E2 -21934.912} C_VEL
LIN {X 0,Y 195.471,Z 843.054,A -85,B 0,C 180,E1 -21939.199,E2 -21939.199} C_VEL
LIN {X 0,Y 196.486,Z 843.289,A -85,B 0,C 180,E1 -21941.221,E2 -21941.221} C_VEL
LIN {X 0,Y 197.835,Z 843.093,A -85,B 0,C 180,E1 -21943.571,E2 -21943.571} C_VEL
LIN {X 0,Y 199.356,Z 842.475,A -85,B 0,C 180,E1 -21945.713,E2 -21945.713} C_VEL
LIN {X 0,Y 201.212,Z 841.29,A -85,B 0,C 180,E1 -21947.96,E2 -21947.96} C_VEL
LIN {X 0,Y 204.252,Z 838.737,A -85,B 0,C 180,E1 -21951.092,E2 -21951.092} C_VEL
LIN {X 0,Y 207.881,Z 834.973,A -85,B 0,C 180,E1 -21954.179,E2 -21954.179} C_VEL
LIN {X 0,Y 212.332,Z 829.564,A -85,B 0,C 180,E1 -21957.352,E2 -21957.352} C_VEL
LIN {X 0,Y 217.206,Z 822.551,A -85,B 0,C 180,E1 -21960.387,E2 -21960.387} C_VEL
LIN {X 0,Y 221.548,Z 815.466,A -85,B 0,C 180,E1 -21962.727,E2 -21962.727} C_VEL
LIN {X 0,Y 222.411,Z 813.947,A -85,B 0,C 180,E1 -21963.17,E2 -21963.17} C_VEL
LIN {X 0,Y 222.92,Z 810.851,A -85,B 0,C 180,E1 -21964.52,E2 -21964.52} C_VEL
LIN {X 0,Y 223.127,Z 806.614,A -85,B 0,C 180,E1 -21966.463,E2 -21966.463} C_VEL
LIN {X 0,Y 222.136,Z 799.99,A -85,B 0,C 180,E1 -21970.022,E2 -21970.022} C_VEL
LIN {X 0,Y 221.135,Z 795.166,A -85,B 0,C 180,E1 -21972.854,E2 -21972.854} C_VEL
LIN {X 0,Y 219.975,Z 792.739,A -85,B 0,C 180,E1 -21974.809,E2 -21974.809} C_VEL
LIN {X 0,Y 217.436,Z 789.634,A -85,B 0,C 180,E1 -21978.858,E2 -21978.858} C_VEL
LIN {X 0,Y 216.39,Z 788.595,A -85,B 0,C 180,E1 -21980.932,E2 -21980.932} C_VEL
LIN {X 0,Y 214.675,Z 788.095,A -85,B 0,C 180,E1 -21985.188,E2 -21985.188} C_VEL
LIN {X 0,Y 214.32,Z 788.279,A -85,B 0,C 180,E1 -21987.7,E2 -21987.7} C_VEL
LIN {X 0,Y 214.139,Z 789.052,A -85,B 0,C 180,E1 -21989.492,E2 -21989.492} C_VEL
LIN {X 0,Y 214.507,Z 792.219,A -85,B 0,C 180,E1 -21993.847,E2 -21993.847} C_VEL
LIN {X 0,Y 214.92,Z 794.909,A -85,B 0,C 180,E1 -21996.058,E2 -21996.058} C_VEL
LIN {X 0,Y 216.61,Z 801.737,A -85,B 0,C 180,E1 -22000.459,E2 -22000.459} C_VEL
LIN {X 0,Y 218.216,Z 808.93,A -85,B 0,C 180,E1 -22003.868,E2 -22003.868} C_VEL
LIN {X 0,Y 218.514,Z 811.868,A -85,B 0,C 180,E1 -22004.961,E2 -22004.961} C_VEL
LIN {X 0,Y 217.583,Z 823.024,A -85,B 0,C 180,E1 -22007.98,E2 -22007.98} C_VEL
LIN {X 0,Y 216.133,Z 833.142,A -85,B 0,C 180,E1 -22010.649,E2 -22010.649} C_VEL
LIN {X 0,Y 213.913,Z 843.182,A -85,B 0,C 180,E1 -22013.328,E2 -22013.328} C_VEL
LIN {X 0,Y 210.719,Z 853.36,A -85,B 0,C 180,E1 -22016.196,E2 -22016.196} C_VEL
LIN {X 0,Y 207.13,Z 861.818,A -85,B 0,C 180,E1 -22018.839,E2 -22018.839} C_VEL
LIN {X 0,Y 203.017,Z 870.607,A -85,B 0,C 180,E1 -22022.138,E2 -22022.138} C_VEL
LIN {X 0,Y 199.575,Z 876.864,A -85,B 0,C 180,E1 -22025.002,E2 -22025.002} C_VEL
LIN {X 0,Y 196.477,Z 882.04,A -85,B 0,C 180,E1 -22027.939,E2 -22027.939} C_VEL
LIN {X 0,Y 194.134,Z 886.283,A -85,B 0,C 180,E1 -22030.985,E2 -22030.985} C_VEL
LIN {X 0,Y 192.189,Z 890.614,A -85,B 0,C 180,E1 -22035.168,E2 -22035.168} C_VEL
LIN {X 0,Y 191.406,Z 893.469,A -85,B 0,C 180,E1 -22039.556,E2 -22039.556} C_VEL
LIN {X 0,Y 190.76,Z 894.128,A -85,B 0,C 180,E1 -22041.31,E2 -22041.31} C_VEL
LIN {X 0,Y 189.351,Z 894.339,A -85,B 0,C 180,E1 -22043.052,E2 -22043.052} C_VEL
LIN {X 0,Y 186.348,Z 893.747,A -85,B 0,C 180,E1 -22046.587,E2 -22046.587} C_VEL
LIN {X 0,Y 185.8,Z 893.134,A -85,B 0,C 180,E1 -22048.407,E2 -22048.407} C_VEL
LIN {X 0,Y 185.894,Z 892.855,A -85,B 0,C 180,E1 -22049.017,E2 -22049.017} C_VEL
LIN {X 0,Y 186.209,Z 892.499,A -85,B 0,C 180,E1 -22050,E2 -22050} C_VEL
LIN {X 0,Y 185.889,Z 891.085,A -85,B 0,C 180,E1 -22052.167,E2 -22052.167} C_VEL
LIN {X 0,Y 185.491,Z 888.001,A -85,B 0,C 180,E1 -22055.435,E2 -22055.435} C_VEL
LIN {X 0,Y 185.2,Z 883.716,A -85,B 0,C 180,E1 -22058.731,E2 -22058.731} C_VEL
LIN {X 0,Y 185.418,Z 877.068,A -85,B 0,C 180,E1 -22062.588,E2 -22062.588} C_VEL
LIN {X 0,Y 186.264,Z 869.828,A -85,B 0,C 180,E1 -22065.876,E2 -22065.876} C_VEL
LIN {X 0,Y 187.502,Z 862.485,A -85,B 0,C 180,E1 -22068.578,E2 -22068.578} C_VEL
LIN {X 0,Y 188.362,Z 856.24,A -85,B 0,C 180,E1 -22070.503,E2 -22070.503} C_VEL
LIN {X 0,Y 188.519,Z 846.508,A -85,B 0,C 180,E1 -22073.044,E2 -22073.044} C_VEL
LIN {X 0,Y 188.483,Z 835.648,A -85,B 0,C 180,E1 -22075.392,E2 -22075.392} C_VEL
LIN {X 0,Y 188.407,Z 823.627,A -85,B 0,C 180,E1 -22077.491,E2 -22077.491} C_VEL
LIN {X 0,Y 188.005,Z 811.085,A -85,B 0,C 180,E1 -22079.251,E2 -22079.251} C_VEL
LIN {X 0,Y 187.465,Z 798.028,A -85,B 0,C 180,E1 -22080.665,E2 -22080.665} C_VEL
LIN {X 0,Y 187.01,Z 788.233,A -85,B 0,C 180,E1 -22081.485,E2 -22081.485} C_VEL
LIN {X 0,Y 189.415,Z 778.897,A -85,B 0,C 180,E1 -22087.75,E2 -22087.75} C_VEL
LIN {X 0,Y 189.942,Z 777.003,A -85,B 0,C 180,E1 -22089.012,E2 -22089.012} C_VEL
LIN {X 0,Y 190.032,Z 775.089,A -85,B 0,C 180,E1 -22090.33,E2 -22090.33} C_VEL
LIN {X 0,Y 188.56,Z 768.44,A -85,B 0,C 180,E1 -22095.086,E2 -22095.086} C_VEL
LIN {X 0,Y 187.162,Z 761.484,A -85,B 0,C 180,E1 -22100.331,E2 -22100.331} C_VEL
LIN {X 0,Y 185.961,Z 755.05,A -85,B 0,C 180,E1 -22105.466,E2 -22105.466} C_VEL
LIN {X 0,Y 185.638,Z 753.36,A -85,B 0,C 180,E1 -22106.875,E2 -22106.875} C_VEL
LIN {X 0,Y 185.583,Z 753.365,A -85,B 0,C 180,E1 -22110.576,E2 -22110.576} C_VEL
LIN {X 0,Y 185.581,Z 753.366,A -85,B 0,C 180,E1 -22115.382,E2 -22115.382} C_VEL
LIN {X 0,Y 185.675,Z 753.351,A -85,B 0,C 180,E1 -22121.134,E2 -22121.134} C_VEL
LIN {X 0,Y 185.697,Z 753.353,A -85,B 0,C 180,E1 -22124.638,E2 -22124.638} C_VEL
LIN {X 0,Y 185.89,Z 753.325,A -85,B 0,C 180,E1 -22129.418,E2 -22129.418} C_VEL
LIN {X 0,Y 185.946,Z 753.321,A -85,B 0,C 180,E1 -22133.49,E2 -22133.49} C_VEL
LIN {X 0,Y 186.203,Z 753.287,A -85,B 0,C 180,E1 -22137.837,E2 -22137.837} C_VEL
LIN {X 0,Y 186.403,Z 753.261,A -85,B 0,C 180,E1 -22140,E2 -22140} C_VEL
LIN {X 0,Y 185.911,Z 753.326,A -85,B 0,C 180,E1 -22144.336,E2 -22144.336} C_VEL
LIN {X 0,Y 185.976,Z 753.315,A -85,B 0,C 180,E1 -22148.694,E2 -22148.694} C_VEL
LIN {X 0,Y 185.722,Z 753.351,A -85,B 0,C 180,E1 -22153.124,E2 -22153.124} C_VEL
LIN {X 0,Y 185.685,Z 753.353,A -85,B 0,C 180,E1 -22157.626,E2 -22157.626} C_VEL
LIN {X 0,Y 185.556,Z 753.369,A -85,B 0,C 180,E1 -22162.257,E2 -22162.257} C_VEL
LIN {X 0,Y 185.5,Z 753.376,A -85,B 0,C 180,E1 -22167.042,E2 -22167.042} C_VEL
LIN {X 0,Y 185.544,Z 753.374,A -85,B 0,C 180,E1 -22169.5,E2 -22169.5} C_VEL
LIN {X 0,Y 185.497,Z 753.374,A -85,B 0,C 180,E1 -22174.633,E2 -22174.633} C_VEL
LIN {X 0,Y 185.5,Z 753.377,A -85,B 0,C 180,E1 -22177.315,E2 -22177.315} C_VEL
LIN {X 0,Y 185.461,Z 753.379,A -85,B 0,C 180,E1 -22180.721,E2 -22180.721} C_VEL
LIN {X 0,Y 185.456,Z 753.385,A -85,B 0,C 180,E1 -22186.057,E2 -22186.057} C_VEL
LIN {X 0,Y 185.456,Z 753.382,A -85,B 0,C 180,E1 -22189.892,E2 -22189.892} C_VEL
LIN {X 0,Y 185.501,Z 753.376,A -85,B 0,C 180,E1 -22192.714,E2 -22192.714} C_VEL
LIN {X 0,Y 185.531,Z 753.373,A -85,B 0,C 180,E1 -22197.973,E2 -22197.973} C_VEL
LIN {X 0,Y 185.494,Z 753.378,A -85,B 0,C 180,E1 -22202.957,E2 -22202.957} C_VEL
LIN {X 0,Y 185.554,Z 753.367,A -85,B 0,C 180,E1 -22207.743,E2 -22207.743} C_VEL
LIN {X 0,Y 185.658,Z 753.358,A -85,B 0,C 180,E1 -22212.372,E2 -22212.372} C_VEL
LIN {X 0,Y 185.719,Z 753.347,A -85,B 0,C 180,E1 -22216.877,E2 -22216.877} C_VEL
LIN {X 0,Y 185.976,Z 753.319,A -85,B 0,C 180,E1 -22221.306,E2 -22221.306} C_VEL
LIN {X 0,Y 186.178,Z 753.291,A -85,B 0,C 180,E1 -22227.837,E2 -22227.837} C_VEL
LIN {X 0,Y 186.382,Z 753.267,A -85,B 0,C 180,E1 -22230,E2 -22230} C_VEL
LIN {X 0,Y 185.888,Z 753.323,A -85,B 0,C 180,E1 -22234.337,E2 -22234.337} C_VEL
LIN {X 0,Y 185.977,Z 753.318,A -85,B 0,C 180,E1 -22238.694,E2 -22238.694} C_VEL
LIN {X 0,Y 185.731,Z 753.345,A -85,B 0,C 180,E1 -22243.123,E2 -22243.123} C_VEL
LIN {X 0,Y 185.693,Z 753.356,A -85,B 0,C 180,E1 -22247.625,E2 -22247.625} C_VEL
LIN {X 0,Y 185.581,Z 753.368,A -85,B 0,C 180,E1 -22252.254,E2 -22252.254} C_VEL
LIN {X 0,Y 185.511,Z 753.376,A -85,B 0,C 180,E1 -22257.041,E2 -22257.041} C_VEL
LIN {X 0,Y 185.545,Z 753.374,A -85,B 0,C 180,E1 -22262.025,E2 -22262.025} C_VEL
LIN {X 0,Y 185.58,Z 753.368,A -85,B 0,C 180,E1 -22262.873,E2 -22262.873} C_VEL
LIN {X 0,Y 190.084,Z 768.088,A -85,B 0,C 180,E1 -22265.387,E2 -22265.387} C_VEL
LIN {X 0,Y 193.039,Z 779.104,A -85,B 0,C 180,E1 -22267.577,E2 -22267.577} C_VEL
LIN {X 0,Y 194.208,Z 783.839,A -85,B 0,C 180,E1 -22268.627,E2 -22268.627} C_VEL
LIN {X 0,Y 192.365,Z 795.249,A -85,B 0,C 180,E1 -22271.12,E2 -22271.12} C_VEL
LIN {X 0,Y 190.701,Z 804.965,A -85,B 0,C 180,E1 -22273.73,E2 -22273.73} C_VEL
LIN {X 0,Y 189.184,Z 813.618,A -85,B 0,C 180,E1 -22276.586,E2 -22276.586} C_VEL
LIN {X 0,Y 187.845,Z 821.785,A -85,B 0,C 180,E1 -22279.902,E2 -22279.902} C_VEL
LIN {X 0,Y 186.973,Z 828.026,A -85,B 0,C 180,E1 -22283.028,E2 -22283.028} C_VEL
LIN {X 0,Y 186.489,Z 832.853,A -85,B 0,C 180,E1 -22286.006,E2 -22286.006} C_VEL
LIN {X 0,Y 186.277,Z 837.063,A -85,B 0,C 180,E1 -22289.266,E2 -22289.266} C_VEL
LIN {X 0,Y 186.557,Z 840.795,A -85,B 0,C 180,E1 -22293.123,E2 -22293.123} C_VEL
LIN {X 0,Y 187.115,Z 842.464,A -85,B 0,C 180,E1 -22295.596,E2 -22295.596} C_VEL
LIN {X 0,Y 188.292,Z 843.939,A -85,B 0,C 180,E1 -22298.929,E2 -22298.929} C_VEL
LIN {X 0,Y 190.66,Z 844.458,A -85,B 0,C 180,E1 -22303.416,E2 -22303.416} C_VEL
LIN {X 0,Y 193.6,Z 843.379,A -85,B 0,C 180,E1 -22307.419,E2 -22307.419} C_VEL
LIN {X 0,Y 195.632,Z 842.124,A -85,B 0,C 180,E1 -22309.652,E2 -22309.652} C_VEL
LIN {X 0,Y 198.523,Z 839.801,A -85,B 0,C 180,E1 -22312.415,E2 -22312.415} C_VEL
LIN {X 0,Y 203.161,Z 835.33,A -85,B 0,C 180,E1 -22316.033,E2 -22316.033} C_VEL
LIN {X 0,Y 208.394,Z 829.07,A -85,B 0,C 180,E1 -22319.517,E2 -22319.517} C_VEL
LIN {X 0,Y 213.418,Z 822.116,A -85,B 0,C 180,E1 -22322.359,E2 -22322.359} C_VEL
LIN {X 0,Y 216.993,Z 816.535,A -85,B 0,C 180,E1 -22324.179,E2 -22324.179} C_VEL
LIN {X 0,Y 217.734,Z 811.792,A -85,B 0,C 180,E1 -22326.487,E2 -22326.487} C_VEL
LIN {X 0,Y 217.524,Z 806.846,A -85,B 0,C 180,E1 -22329.296,E2 -22329.296} C_VEL
LIN {X 0,Y 216.98,Z 802.115,A -85,B 0,C 180,E1 -22332.154,E2 -22332.154} C_VEL
LIN {X 0,Y 216.669,Z 800.441,A -85,B 0,C 180,E1 -22333.318,E2 -22333.318} C_VEL
LIN {X 0,Y 215.813,Z 798.418,A -85,B 0,C 180,E1 -22335.101,E2 -22335.101} C_VEL
LIN {X 0,Y 213.7,Z 795.597,A -85,B 0,C 180,E1 -22339.2,E2 -22339.2} C_VEL
LIN {X 0,Y 212.391,Z 794.644,A -85,B 0,C 180,E1 -22342.101,E2 -22342.101} C_VEL
LIN {X 0,Y 211.343,Z 794.462,A -85,B 0,C 180,E1 -22346.121,E2 -22346.121} C_VEL
LIN {X 0,Y 211.159,Z 794.712,A -85,B 0,C 180,E1 -22347.772,E2 -22347.772} C_VEL
LIN {X 0,Y 210.999,Z 797.367,A -85,B 0,C 180,E1 -22352.204,E2 -22352.204} C_VEL
LIN {X 0,Y 211.375,Z 799.346,A -85,B 0,C 180,E1 -22354.418,E2 -22354.418} C_VEL
LIN {X 0,Y 212.779,Z 807.645,A -85,B 0,C 180,E1 -22360.098,E2 -22360.098} C_VEL
LIN {X 0,Y 213.968,Z 815.15,A -85,B 0,C 180,E1 -22363.729,E2 -22363.729} C_VEL
LIN {X 0,Y 213.246,Z 821.334,A -85,B 0,C 180,E1 -22365.59,E2 -22365.59} C_VEL
LIN {X 0,Y 211.665,Z 831.166,A -85,B 0,C 180,E1 -22368.389,E2 -22368.389} C_VEL
LIN {X 0,Y 209.074,Z 841.892,A -85,B 0,C 180,E1 -22371.421,E2 -22371.421} C_VEL
LIN {X 0,Y 205.628,Z 852.187,A -85,B 0,C 180,E1 -22374.476,E2 -22374.476} C_VEL
LIN {X 0,Y 202.417,Z 859.559,A -85,B 0,C 180,E1 -22376.849,E2 -22376.849} C_VEL
LIN {X 0,Y 197.885,Z 868.423,A -85,B 0,C 180,E1 -22380.183,E2 -22380.183} C_VEL
LIN {X 0,Y 194.384,Z 874.767,A -85,B 0,C 180,E1 -22383.131,E2 -22383.131} C_VEL
LIN {X 0,Y 190.869,Z 880.095,A -85,B 0,C 180,E1 -22386.106,E2 -22386.106} C_VEL
LIN {X 0,Y 187.369,Z 885.73,A -85,B 0,C 180,E1 -22390.27,E2 -22390.27} C_VEL
LIN {X 0,Y 185.269,Z 889.792,A -85,B 0,C 180,E1 -22394.601,E2 -22394.601} C_VEL
LIN {X 0,Y 184.381,Z 892.433,A -85,B 0,C 180,E1 -22399.013,E2 -22399.013} C_VEL
LIN {X 0,Y 184.69,Z 893.663,A -85,B 0,C 180,E1 -22403.445,E2 -22403.445} C_VEL
LIN {X 0,Y 185.588,Z 893.284,A -85,B 0,C 180,E1 -22407.83,E2 -22407.83} C_VEL
LIN {X 0,Y 185.894,Z 892.855,A -85,B 0,C 180,E1 -22409.017,E2 -22409.017} C_VEL
LIN {X 0,Y 185.822,Z 892.319,A -85,B 0,C 180,E1 -22410.206,E2 -22410.206} C_VEL
LIN {X 0,Y 185.094,Z 891.462,A -85,B 0,C 180,E1 -22411.368,E2 -22411.368} C_VEL
LIN {X 0,Y 182.537,Z 889.21,A -85,B 0,C 180,E1 -22413.609,E2 -22413.609} C_VEL
LIN {X 0,Y 179.701,Z 886.344,A -85,B 0,C 180,E1 -22415.868,E2 -22415.868} C_VEL
LIN {X 0,Y 178.387,Z 883.935,A -85,B 0,C 180,E1 -22417.613,E2 -22417.613} C_VEL
LIN {X 0,Y 178.243,Z 883.085,A -85,B 0,C 180,E1 -22418.207,E2 -22418.207} C_VEL
LIN {X 0,Y 178.328,Z 877.162,A -85,B 0,C 180,E1 -22421.941,E2 -22421.941} C_VEL
LIN {X 0,Y 179.045,Z 870.169,A -85,B 0,C 180,E1 -22425.364,E2 -22425.364} C_VEL
LIN {X 0,Y 180.502,Z 861.54,A -85,B 0,C 180,E1 -22428.737,E2 -22428.737} C_VEL
LIN {X 0,Y 181.247,Z 856.38,A -85,B 0,C 180,E1 -22430.425,E2 -22430.425} C_VEL
LIN {X 0,Y 181.442,Z 845.549,A -85,B 0,C 180,E1 -22433.392,E2 -22433.392} C_VEL
LIN {X 0,Y 181.419,Z 835.132,A -85,B 0,C 180,E1 -22435.746,E2 -22435.746} C_VEL
LIN {X 0,Y 181.361,Z 822.701,A -85,B 0,C 180,E1 -22438.025,E2 -22438.025} C_VEL
LIN {X 0,Y 180.962,Z 809.118,A -85,B 0,C 180,E1 -22440.001,E2 -22440.001} C_VEL
LIN {X 0,Y 180.481,Z 795.358,A -85,B 0,C 180,E1 -22441.497,E2 -22441.497} C_VEL
LIN {X 0,Y 180.135,Z 787.281,A -85,B 0,C 180,E1 -22442.207,E2 -22442.207} C_VEL
LIN {X 0,Y 182.729,Z 777.694,A -85,B 0,C 180,E1 -22448.894,E2 -22448.894} C_VEL
LIN {X 0,Y 182.82,Z 774.992,A -85,B 0,C 180,E1 -22450.807,E2 -22450.807} C_VEL
LIN {X 0,Y 181.041,Z 767.035,A -85,B 0,C 180,E1 -22456.803,E2 -22456.803} C_VEL
LIN {X 0,Y 179.909,Z 761.261,A -85,B 0,C 180,E1 -22461.378,E2 -22461.378} C_VEL
LIN {X 0,Y 178.742,Z 755.008,A -85,B 0,C 180,E1 -22466.601,E2 -22466.601} C_VEL
LIN {X 0,Y 178.568,Z 754.242,A -85,B 0,C 180,E1 -22467.404,E2 -22467.404} C_VEL
LIN {X 0,Y 178.488,Z 754.249,A -85,B 0,C 180,E1 -22471.803,E2 -22471.803} C_VEL
LIN {X 0,Y 178.5,Z 754.249,A -85,B 0,C 180,E1 -22476.814,E2 -22476.814} C_VEL
LIN {X 0,Y 178.651,Z 754.226,A -85,B 0,C 180,E1 -22481.657,E2 -22481.657} C_VEL
LIN {X 0,Y 178.66,Z 754.231,A -85,B 0,C 180,E1 -22486.348,E2 -22486.348} C_VEL
LIN {X 0,Y 178.913,Z 754.195,A -85,B 0,C 180,E1 -22490.96,E2 -22490.96} C_VEL
LIN {X 0,Y 179.149,Z 754.165,A -85,B 0,C 180,E1 -22497.752,E2 -22497.752} C_VEL
LIN {X 0,Y 179.367,Z 754.137,A -85,B 0,C 180,E1 -22500,E2 -22500} C_VEL
LIN {X 0,Y 178.858,Z 754.206,A -85,B 0,C 180,E1 -22504.508,E2 -22504.508} C_VEL
LIN {X 0,Y 178.906,Z 754.197,A -85,B 0,C 180,E1 -22509.041,E2 -22509.041} C_VEL
LIN {X 0,Y 178.65,Z 754.229,A -85,B 0,C 180,E1 -22513.653,E2 -22513.653} C_VEL
LIN {X 0,Y 178.609,Z 754.237,A -85,B 0,C 180,E1 -22519.202,E2 -22519.202} C_VEL
LIN {X 0,Y 178.466,Z 754.25,A -85,B 0,C 180,E1 -22525.077,E2 -22525.077} C_VEL
LIN {X 0,Y 178.461,Z 754.253,A -85,B 0,C 180,E1 -22530.795,E2 -22530.795} C_VEL
LIN {X 0,Y 178.483,Z 754.248,A -85,B 0,C 180,E1 -22534.218,E2 -22534.218} C_VEL
LIN {X 0,Y 178.387,Z 754.263,A -85,B 0,C 180,E1 -22539.077,E2 -22539.077} C_VEL
LIN {X 0,Y 178.393,Z 754.259,A -85,B 0,C 180,E1 -22542.047,E2 -22542.047} C_VEL
LIN {X 0,Y 178.392,Z 754.261,A -85,B 0,C 180,E1 -22545.165,E2 -22545.165} C_VEL
LIN {X 0,Y 178.398,Z 754.261,A -85,B 0,C 180,E1 -22548.462,E2 -22548.462} C_VEL
LIN {X 0,Y 178.42,Z 754.259,A -85,B 0,C 180,E1 -22553.782,E2 -22553.782} C_VEL
LIN {X 0,Y 178.485,Z 754.251,A -85,B 0,C 180,E1 -22556.546,E2 -22556.546} C_VEL
LIN {X 0,Y 178.425,Z 754.257,A -85,B 0,C 180,E1 -22561.792,E2 -22561.792} C_VEL
LIN {X 0,Y 178.469,Z 754.251,A -85,B 0,C 180,E1 -22566.809,E2 -22566.809} C_VEL
LIN {X 0,Y 178.613,Z 754.234,A -85,B 0,C 180,E1 -22571.653,E2 -22571.653} C_VEL
LIN {X 0,Y 178.646,Z 754.229,A -85,B 0,C 180,E1 -22576.347,E2 -22576.347} C_VEL
LIN {X 0,Y 178.907,Z 754.201,A -85,B 0,C 180,E1 -22580.96,E2 -22580.96} C_VEL
LIN {X 0,Y 179.126,Z 754.17,A -85,B 0,C 180,E1 -22587.752,E2 -22587.752} C_VEL
LIN {X 0,Y 179.347,Z 754.143,A -85,B 0,C 180,E1 -22590,E2 -22590} C_VEL
LIN {X 0,Y 178.837,Z 754.201,A -85,B 0,C 180,E1 -22594.508,E2 -22594.508} C_VEL
LIN {X 0,Y 178.907,Z 754.199,A -85,B 0,C 180,E1 -22599.041,E2 -22599.041} C_VEL
LIN {X 0,Y 178.66,Z 754.227,A -85,B 0,C 180,E1 -22603.652,E2 -22603.652} C_VEL
LIN {X 0,Y 178.625,Z 754.234,A -85,B 0,C 180,E1 -22609.215,E2 -22609.215} C_VEL
LIN {X 0,Y 178.518,Z 754.246,A -85,B 0,C 180,E1 -22615.111,E2 -22615.111} C_VEL
LIN {X 0,Y 178.468,Z 754.254,A -85,B 0,C 180,E1 -22620.793,E2 -22620.793} C_VEL
LIN {X 0,Y 178.51,Z 754.25,A -85,B 0,C 180,E1 -22622.191,E2 -22622.191} C_VEL
LIN {X 0,Y 182.371,Z 766.662,A -85,B 0,C 180,E1 -22624.37,E2 -22624.37} C_VEL
LIN {X 0,Y 185.159,Z 776.615,A -85,B 0,C 180,E1 -22626.365,E2 -22626.365} C_VEL
LIN {X 0,Y 187.222,Z 785.097,A -85,B 0,C 180,E1 -22628.27,E2 -22628.27} C_VEL
LIN {X 0,Y 185.408,Z 795.882,A -85,B 0,C 180,E1 -22630.701,E2 -22630.701} C_VEL
LIN {X 0,Y 183.626,Z 806.127,A -85,B 0,C 180,E1 -22633.546,E2 -22633.546} C_VEL
LIN {X 0,Y 181.93,Z 815.411,A -85,B 0,C 180,E1 -22636.753,E2 -22636.753} C_VEL
LIN {X 0,Y 180.661,Z 823.136,A -85,B 0,C 180,E1 -22640.06,E2 -22640.06} C_VEL
LIN {X 0,Y 179.831,Z 829.496,A -85,B 0,C 180,E1 -22643.416,E2 -22643.416} C_VEL
LIN {X 0,Y 179.32,Z 834.552,A -85,B 0,C 180,E1 -22646.722,E2 -22646.722} C_VEL
LIN {X 0,Y 179.215,Z 839.349,A -85,B 0,C 180,E1 -22650.793,E2 -22650.793} C_VEL
LIN {X 0,Y 179.789,Z 842.524,A -85,B 0,C 180,E1 -22654.533,E2 -22654.533} C_VEL
LIN {X 0,Y 181.092,Z 844.75,A -85,B 0,C 180,E1 -22658.658,E2 -22658.658} C_VEL
LIN {X 0,Y 183.47,Z 845.671,A -85,B 0,C 180,E1 -22663.268,E2 -22663.268} C_VEL
LIN {X 0,Y 186.865,Z 844.872,A -85,B 0,C 180,E1 -22667.924,E2 -22667.924} C_VEL
LIN {X 0,Y 191.391,Z 842.127,A -85,B 0,C 180,E1 -22672.51,E2 -22672.51} C_VEL
LIN {X 0,Y 195.565,Z 838.655,A -85,B 0,C 180,E1 -22675.878,E2 -22675.878} C_VEL
LIN {X 0,Y 200.163,Z 833.989,A -85,B 0,C 180,E1 -22678.994,E2 -22678.994} C_VEL
LIN {X 0,Y 205.182,Z 828.076,A -85,B 0,C 180,E1 -22681.963,E2 -22681.963} C_VEL
LIN {X 0,Y 210.716,Z 820.569,A -85,B 0,C 180,E1 -22684.783,E2 -22684.783} C_VEL
LIN {X 0,Y 211.541,Z 819.206,A -85,B 0,C 180,E1 -22685.242,E2 -22685.242} C_VEL
LIN {X 0,Y 212.392,Z 814.869,A -85,B 0,C 180,E1 -22687.606,E2 -22687.606} C_VEL
LIN {X 0,Y 212.342,Z 808.83,A -85,B 0,C 180,E1 -22691.454,E2 -22691.454} C_VEL
LIN {X 0,Y 212.148,Z 806.026,A -85,B 0,C 180,E1 -22693.409,E2 -22693.409} C_VEL
LIN {X 0,Y 211.447,Z 803.938,A -85,B 0,C 180,E1 -22695.442,E2 -22695.442} C_VEL
LIN {X 0,Y 209.697,Z 801.424,A -85,B 0,C 180,E1 -22699.582,E2 -22699.582} C_VEL
LIN {X 0,Y 208.882,Z 800.76,A -85,B 0,C 180,E1 -22701.722,E2 -22701.722} C_VEL
LIN {X 0,Y 207.869,Z 800.645,A -85,B 0,C 180,E1 -22706.074,E2 -22706.074} C_VEL
LIN {X 0,Y 207.589,Z 801.254,A -85,B 0,C 180,E1 -22708.328,E2 -22708.328} C_VEL
LIN {X 0,Y 207.618,Z 804.143,A -85,B 0,C 180,E1 -22712.793,E2 -22712.793} C_VEL
LIN {X 0,Y 207.782,Z 806.67,A -85,B 0,C 180,E1 -22715.1,E2 -22715.1} C_VEL
LIN {X 0,Y 208.685,Z 813.441,A -85,B 0,C 180,E1 -22719.782,E2 -22719.782} C_VEL
LIN {X 0,Y 209.245,Z 820.071,A -85,B 0,C 180,E1 -22723.084,E2 -22723.084} C_VEL
LIN {X 0,Y 207.183,Z 830.288,A -85,B 0,C 180,E1 -22726.237,E2 -22726.237} C_VEL
LIN {X 0,Y 204.595,Z 840.264,A -85,B 0,C 180,E1 -22729.257,E2 -22729.257} C_VEL
LIN {X 0,Y 201.148,Z 850.057,A -85,B 0,C 180,E1 -22732.306,E2 -22732.306} C_VEL
LIN {X 0,Y 197.246,Z 858.766,A -85,B 0,C 180,E1 -22735.243,E2 -22735.243} C_VEL
LIN {X 0,Y 191.705,Z 868.604,A -85,B 0,C 180,E1 -22739.119,E2 -22739.119} C_VEL
LIN {X 0,Y 188.033,Z 874.713,A -85,B 0,C 180,E1 -22742.147,E2 -22742.147} C_VEL
LIN {X 0,Y 183.318,Z 881.243,A -85,B 0,C 180,E1 -22746.262,E2 -22746.262} C_VEL
LIN {X 0,Y 180.619,Z 885.116,A -85,B 0,C 180,E1 -22749.5,E2 -22749.5} C_VEL
LIN {X 0,Y 178.371,Z 888.986,A -85,B 0,C 180,E1 -22753.99,E2 -22753.99} C_VEL
LIN {X 0,Y 177.376,Z 891.451,A -85,B 0,C 180,E1 -22758.573,E2 -22758.573} C_VEL
LIN {X 0,Y 177.633,Z 892.455,A -85,B 0,C 180,E1 -22763.183,E2 -22763.183} C_VEL
LIN {X 0,Y 178.58,Z 891.969,A -85,B 0,C 180,E1 -22767.744,E2 -22767.744} C_VEL
LIN {X 0,Y 179.217,Z 891.117,A -85,B 0,C 180,E1 -22770,E2 -22770} C_VEL
LIN {X 0,Y 178.717,Z 888.621,A -85,B 0,C 180,E1 -22773.381,E2 -22773.381} C_VEL
LIN {X 0,Y 178.344,Z 884.98,A -85,B 0,C 180,E1 -22776.789,E2 -22776.789} C_VEL
LIN {X 0,Y 178.243,Z 883.085,A -85,B 0,C 180,E1 -22778.207,E2 -22778.207} C_VEL
LIN {X 0,Y 177.534,Z 880.477,A -85,B 0,C 180,E1 -22779.897,E2 -22779.897} C_VEL
LIN {X 0,Y 174.964,Z 875.493,A -85,B 0,C 180,E1 -22782.563,E2 -22782.563} C_VEL
LIN {X 0,Y 172.717,Z 869.876,A -85,B 0,C 180,E1 -22785.169,E2 -22785.169} C_VEL
LIN {X 0,Y 172.537,Z 866.214,A -85,B 0,C 180,E1 -22786.718,E2 -22786.718} C_VEL
LIN {X 0,Y 174.038,Z 857.229,A -85,B 0,C 180,E1 -22790.075,E2 -22790.075} C_VEL
LIN {X 0,Y 174.321,Z 848.459,A -85,B 0,C 180,E1 -22792.736,E2 -22792.736} C_VEL
LIN {X 0,Y 174.425,Z 838.15,A -85,B 0,C 180,E1 -22795.347,E2 -22795.347} C_VEL
LIN {X 0,Y 174.383,Z 825.716,A -85,B 0,C 180,E1 -22797.9,E2 -22797.9} C_VEL
LIN {X 0,Y 174.157,Z 813.269,A -85,B 0,C 180,E1 -22799.959,E2 -22799.959} C_VEL
LIN {X 0,Y 173.749,Z 799.735,A -85,B 0,C 180,E1 -22801.682,E2 -22801.682} C_VEL
LIN {X 0,Y 173.26,Z 786.311,A -85,B 0,C 180,E1 -22802.941,E2 -22802.941} C_VEL
LIN {X 0,Y 175.378,Z 778.843,A -85,B 0,C 180,E1 -22808.399,E2 -22808.399} C_VEL
LIN {X 0,Y 175.808,Z 776.981,A -85,B 0,C 180,E1 -22809.762,E2 -22809.762} C_VEL
LIN {X 0,Y 175.048,Z 772.662,A -85,B 0,C 180,E1 -22813.042,E2 -22813.042} C_VEL
LIN {X 0,Y 173.63,Z 766.32,A -85,B 0,C 180,E1 -22818.097,E2 -22818.097} C_VEL
LIN {X 0,Y 172.382,Z 759.604,A -85,B 0,C 180,E1 -22823.701,E2 -22823.701} C_VEL
LIN {X 0,Y 171.518,Z 755.121,A -85,B 0,C 180,E1 -22827.813,E2 -22827.813} C_VEL
LIN {X 0,Y 171.415,Z 755.126,A -85,B 0,C 180,E1 -22833.192,E2 -22833.192} C_VEL
LIN {X 0,Y 171.454,Z 755.127,A -85,B 0,C 180,E1 -22838.351,E2 -22838.351} C_VEL
LIN {X 0,Y 171.579,Z 755.107,A -85,B 0,C 180,E1 -22840.872,E2 -22840.872} C_VEL
LIN {X 0,Y 171.578,Z 755.112,A -85,B 0,C 180,E1 -22845.773,E2 -22845.773} C_VEL
LIN {X 0,Y 171.849,Z 755.075,A -85,B 0,C 180,E1 -22850.585,E2 -22850.585} C_VEL
LIN {X 0,Y 171.81,Z 755.082,A -85,B 0,C 180,E1 -22855.308,E2 -22855.308} C_VEL
LIN {X 0,Y 172.33,Z 755.013,A -85,B 0,C 180,E1 -22860,E2 -22860} C_VEL
LIN {X 0,Y 171.807,Z 755.085,A -85,B 0,C 180,E1 -22864.693,E2 -22864.693} C_VEL
LIN {X 0,Y 171.845,Z 755.077,A -85,B 0,C 180,E1 -22869.416,E2 -22869.416} C_VEL
LIN {X 0,Y 171.568,Z 755.111,A -85,B 0,C 180,E1 -22874.228,E2 -22874.228} C_VEL
LIN {X 0,Y 171.528,Z 755.119,A -85,B 0,C 180,E1 -22879.546,E2 -22879.546} C_VEL
LIN {X 0,Y 171.404,Z 755.131,A -85,B 0,C 180,E1 -22885.57,E2 -22885.57} C_VEL
LIN {X 0,Y 171.418,Z 755.13,A -85,B 0,C 180,E1 -22890.573,E2 -22890.573} C_VEL
LIN {X 0,Y 171.393,Z 755.131,A -85,B 0,C 180,E1 -22895.035,E2 -22895.035} C_VEL
LIN {X 0,Y 171.343,Z 755.14,A -85,B 0,C 180,E1 -22898.801,E2 -22898.801} C_VEL
LIN {X 0,Y 171.319,Z 755.144,A -85,B 0,C 180,E1 -22904.219,E2 -22904.219} C_VEL
LIN {X 0,Y 171.33,Z 755.14,A -85,B 0,C 180,E1 -22908.98,E2 -22908.98} C_VEL
LIN {X 0,Y 171.36,Z 755.135,A -85,B 0,C 180,E1 -22912.034,E2 -22912.034} C_VEL
LIN {X 0,Y 171.398,Z 755.133,A -85,B 0,C 180,E1 -22915.093,E2 -22915.093} C_VEL
LIN {X 0,Y 171.393,Z 755.132,A -85,B 0,C 180,E1 -22920.524,E2 -22920.524} C_VEL
LIN {X 0,Y 171.406,Z 755.132,A -85,B 0,C 180,E1 -22925.794,E2 -22925.794} C_VEL
LIN {X 0,Y 171.514,Z 755.121,A -85,B 0,C 180,E1 -22930.864,E2 -22930.864} C_VEL
LIN {X 0,Y 171.56,Z 755.11,A -85,B 0,C 180,E1 -22935.772,E2 -22935.772} C_VEL
LIN {X 0,Y 171.845,Z 755.079,A -85,B 0,C 180,E1 -22940.585,E2 -22940.585} C_VEL
LIN {X 0,Y 171.785,Z 755.082,A -85,B 0,C 180,E1 -22945.307,E2 -22945.307} C_VEL
LIN {X 0,Y 172.312,Z 755.02,A -85,B 0,C 180,E1 -22950,E2 -22950} C_VEL
LIN {X 0,Y 171.787,Z 755.08,A -85,B 0,C 180,E1 -22954.694,E2 -22954.694} C_VEL
LIN {X 0,Y 171.845,Z 755.08,A -85,B 0,C 180,E1 -22959.416,E2 -22959.416} C_VEL
LIN {X 0,Y 171.578,Z 755.109,A -85,B 0,C 180,E1 -22964.227,E2 -22964.227} C_VEL
LIN {X 0,Y 171.544,Z 755.116,A -85,B 0,C 180,E1 -22969.559,E2 -22969.559} C_VEL
LIN {X 0,Y 171.446,Z 755.128,A -85,B 0,C 180,E1 -22975.599,E2 -22975.599} C_VEL
LIN {X 0,Y 171.472,Z 755.213,A -85,B 0,C 180,E1 -22981.557,E2 -22981.557} C_VEL
LIN {X 0,Y 175.346,Z 767.662,A -85,B 0,C 180,E1 -22983.788,E2 -22983.788} C_VEL
LIN {X 0,Y 178.234,Z 777.875,A -85,B 0,C 180,E1 -22985.912,E2 -22985.912} C_VEL
LIN {X 0,Y 180.002,Z 785.129,A -85,B 0,C 180,E1 -22987.583,E2 -22987.583} C_VEL
LIN {X 0,Y 180.187,Z 786.841,A -85,B 0,C 180,E1 -22987.994,E2 -22987.994} C_VEL
LIN {X 0,Y 178.208,Z 797.844,A -85,B 0,C 180,E1 -22990.609,E2 -22990.609} C_VEL
LIN {X 0,Y 176.452,Z 807.594,A -85,B 0,C 180,E1 -22993.476,E2 -22993.476} C_VEL
LIN {X 0,Y 174.745,Z 816.895,A -85,B 0,C 180,E1 -22996.865,E2 -22996.865} C_VEL
LIN {X 0,Y 173.449,Z 824.645,A -85,B 0,C 180,E1 -23000.342,E2 -23000.342} C_VEL
LIN {X 0,Y 172.696,Z 830.532,A -85,B 0,C 180,E1 -23003.593,E2 -23003.593} C_VEL
LIN {X 0,Y 172.177,Z 836.771,A -85,B 0,C 180,E1 -23007.951,E2 -23007.951} C_VEL
LIN {X 0,Y 172.268,Z 841.132,A -85,B 0,C 180,E1 -23012.02,E2 -23012.02} C_VEL
LIN {X 0,Y 173.113,Z 844.217,A -85,B 0,C 180,E1 -23016.047,E2 -23016.047} C_VEL
LIN {X 0,Y 174.019,Z 845.594,A -85,B 0,C 180,E1 -23018.686,E2 -23018.686} C_VEL
LIN {X 0,Y 176.257,Z 846.798,A -85,B 0,C 180,E1 -23023.132,E2 -23023.132} C_VEL
LIN {X 0,Y 179.689,Z 846.457,A -85,B 0,C 180,E1 -23027.907,E2 -23027.907} C_VEL
LIN {X 0,Y 184.261,Z 844.299,A -85,B 0,C 180,E1 -23032.607,E2 -23032.607} C_VEL
LIN {X 0,Y 187.967,Z 841.678,A -85,B 0,C 180,E1 -23035.711,E2 -23035.711} C_VEL
LIN {X 0,Y 192.707,Z 837.654,A -85,B 0,C 180,E1 -23038.955,E2 -23038.955} C_VEL
LIN {X 0,Y 197.787,Z 832.419,A -85,B 0,C 180,E1 -23042.036,E2 -23042.036} C_VEL
LIN {X 0,Y 203.618,Z 825.466,A -85,B 0,C 180,E1 -23045.049,E2 -23045.049} C_VEL
LIN {X 0,Y 205.393,Z 823.118,A -85,B 0,C 180,E1 -23045.892,E2 -23045.892} C_VEL
LIN {X 0,Y 206.376,Z 821.144,A -85,B 0,C 180,E1 -23046.845,E2 -23046.845} C_VEL
LIN {X 0,Y 207.043,Z 817.988,A -85,B 0,C 180,E1 -23048.786,E2 -23048.786} C_VEL
LIN {X 0,Y 207.374,Z 812.46,A -85,B 0,C 180,E1 -23052.726,E2 -23052.726} C_VEL
LIN {X 0,Y 207.371,Z 811.155,A -85,B 0,C 180,E1 -23053.723,E2 -23053.723} C_VEL
LIN {X 0,Y 206.887,Z 809.31,A -85,B 0,C 180,E1 -23055.769,E2 -23055.769} C_VEL
LIN {X 0,Y 205.448,Z 807.099,A -85,B 0,C 180,E1 -23060.004,E2 -23060.004} C_VEL
LIN {X 0,Y 204.789,Z 806.653,A -85,B 0,C 180,E1 -23062.179,E2 -23062.179} C_VEL
LIN {X 0,Y 203.98,Z 806.818,A -85,B 0,C 180,E1 -23066.609,E2 -23066.609} C_VEL
LIN {X 0,Y 203.728,Z 808.529,A -85,B 0,C 180,E1 -23070.409,E2 -23070.409} C_VEL
LIN {X 0,Y 203.837,Z 810.954,A -85,B 0,C 180,E1 -23073.481,E2 -23073.481} C_VEL
LIN {X 0,Y 204.257,Z 818.513,A -85,B 0,C 180,E1 -23079.151,E2 -23079.151} C_VEL
LIN {X 0,Y 204.427,Z 822.711,A -85,B 0,C 180,E1 -23081.436,E2 -23081.436} C_VEL
LIN {X 0,Y 204.345,Z 824.642,A -85,B 0,C 180,E1 -23082.331,E2 -23082.331} C_VEL
LIN {X 0,Y 201.515,Z 835.131,A -85,B 0,C 180,E1 -23085.771,E2 -23085.771} C_VEL
LIN {X 0,Y 197.836,Z 845.766,A -85,B 0,C 180,E1 -23089.23,E2 -23089.23} C_VEL
LIN {X 0,Y 193.559,Z 855.361,A -85,B 0,C 180,E1 -23092.542,E2 -23092.542} C_VEL
LIN {X 0,Y 189.931,Z 861.909,A -85,B 0,C 180,E1 -23095.002,E2 -23095.002} C_VEL
LIN {X 0,Y 184.949,Z 869.811,A -85,B 0,C 180,E1 -23098.5,E2 -23098.5} C_VEL
LIN {X 0,Y 180.453,Z 876.325,A -85,B 0,C 180,E1 -23102.137,E2 -23102.137} C_VEL
LIN {X 0,Y 175.767,Z 882.165,A -85,B 0,C 180,E1 -23106.431,E2 -23106.431} C_VEL
LIN {X 0,Y 173.221,Z 885.558,A -85,B 0,C 180,E1 -23109.826,E2 -23109.826} C_VEL
LIN {X 0,Y 171.499,Z 888.178,A -85,B 0,C 180,E1 -23113.33,E2 -23113.33} C_VEL
LIN {X 0,Y 170.396,Z 890.4,A -85,B 0,C 180,E1 -23118.098,E2 -23118.098} C_VEL
LIN {X 0,Y 170.576,Z 891.249,A -85,B 0,C 180,E1 -23122.9,E2 -23122.9} C_VEL
LIN {X 0,Y 171.566,Z 890.607,A -85,B 0,C 180,E1 -23127.652,E2 -23127.652} C_VEL
LIN {X 0,Y 172.244,Z 889.652,A -85,B 0,C 180,E1 -23130,E2 -23130} C_VEL
LIN {X 0,Y 171.723,Z 887.027,A -85,B 0,C 180,E1 -23133.519,E2 -23133.519} C_VEL
LIN {X 0,Y 171.325,Z 883.224,A -85,B 0,C 180,E1 -23137.069,E2 -23137.069} C_VEL
LIN {X 0,Y 171.275,Z 877.258,A -85,B 0,C 180,E1 -23141.179,E2 -23141.179} C_VEL
LIN {X 0,Y 171.894,Z 870.494,A -85,B 0,C 180,E1 -23144.805,E2 -23144.805} C_VEL
LIN {X 0,Y 172.537,Z 866.214,A -85,B 0,C 180,E1 -23146.718,E2 -23146.718} C_VEL
LIN {X 0,Y 172.358,Z 862.423,A -85,B 0,C 180,E1 -23148.207,E2 -23148.207} C_VEL
LIN {X 0,Y 171.216,Z 858.425,A -85,B 0,C 180,E1 -23149.632,E2 -23149.632} C_VEL
LIN {X 0,Y 168.18,Z 849.967,A -85,B 0,C 180,E1 -23152.35,E2 -23152.35} C_VEL
LIN {X 0,Y 167.35,Z 845.42,A -85,B 0,C 180,E1 -23153.669,E2 -23153.669} C_VEL
LIN {X 0,Y 167.313,Z 843.831,A -85,B 0,C 180,E1 -23154.099,E2 -23154.099} C_VEL
LIN {X 0,Y 167.315,Z 832.643,A -85,B 0,C 180,E1 -23156.843,E2 -23156.843} C_VEL
LIN {X 0,Y 167.304,Z 821.468,A -85,B 0,C 180,E1 -23159.073,E2 -23159.073} C_VEL
LIN {X 0,Y 167.1,Z 808.083,A -85,B 0,C 180,E1 -23161.206,E2 -23161.206} C_VEL
LIN {X 0,Y 166.724,Z 794.53,A -85,B 0,C 180,E1 -23162.852,E2 -23162.852} C_VEL
LIN {X 0,Y 166.386,Z 785.302,A -85,B 0,C 180,E1 -23163.76,E2 -23163.76} C_VEL
LIN {X 0,Y 168.358,Z 778.727,A -85,B 0,C 180,E1 -23168.768,E2 -23168.768} C_VEL
LIN {X 0,Y 168.725,Z 777.189,A -85,B 0,C 180,E1 -23169.951,E2 -23169.951} C_VEL
LIN {X 0,Y 167.923,Z 773.075,A -85,B 0,C 180,E1 -23173.227,E2 -23173.227} C_VEL
LIN {X 0,Y 166.283,Z 765.503,A -85,B 0,C 180,E1 -23179.532,E2 -23179.532} C_VEL
LIN {X 0,Y 165.084,Z 759.21,A -85,B 0,C 180,E1 -23185.101,E2 -23185.101} C_VEL
LIN {X 0,Y 164.462,Z 756,A -85,B 0,C 180,E1 -23188.131,E2 -23188.131} C_VEL
LIN {X 0,Y 164.407,Z 756.003,A -85,B 0,C 180,E1 -23194.693,E2 -23194.693} C_VEL
LIN {X 0,Y 164.485,Z 755.994,A -85,B 0,C 180,E1 -23200.052,E2 -23200.052} C_VEL
LIN {X 0,Y 164.525,Z 755.989,A -85,B 0,C 180,E1 -23205.15,E2 -23205.15} C_VEL
LIN {X 0,Y 164.769,Z 755.956,A -85,B 0,C 180,E1 -23210.177,E2 -23210.177} C_VEL
LIN {X 0,Y 164.831,Z 755.953,A -85,B 0,C 180,E1 -23212.651,E2 -23212.651} C_VEL
LIN {X 0,Y 165.044,Z 755.922,A -85,B 0,C 180,E1 -23217.56,E2 -23217.56} C_VEL
LIN {X 0,Y 165.293,Z 755.89,A -85,B 0,C 180,E1 -23220,E2 -23220} C_VEL
LIN {X 0,Y 164.755,Z 755.962,A -85,B 0,C 180,E1 -23224.894,E2 -23224.894} C_VEL
LIN {X 0,Y 164.824,Z 755.948,A -85,B 0,C 180,E1 -23227.35,E2 -23227.35} C_VEL
LIN {X 0,Y 164.703,Z 755.97,A -85,B 0,C 180,E1 -23231.06,E2 -23231.06} C_VEL
LIN {X 0,Y 164.472,Z 755.995,A -85,B 0,C 180,E1 -23237.405,E2 -23237.405} C_VEL
LIN {X 0,Y 164.452,Z 755.999,A -85,B 0,C 180,E1 -23239.992,E2 -23239.992} C_VEL
LIN {X 0,Y 164.339,Z 756.01,A -85,B 0,C 180,E1 -23246.095,E2 -23246.095} C_VEL
LIN {X 0,Y 164.354,Z 756.012,A -85,B 0,C 180,E1 -23251.215,E2 -23251.215} C_VEL
LIN {X 0,Y 164.28,Z 756.02,A -85,B 0,C 180,E1 -23256.794,E2 -23256.794} C_VEL
LIN {X 0,Y 164.286,Z 756.019,A -85,B 0,C 180,E1 -23259.918,E2 -23259.918} C_VEL
LIN {X 0,Y 164.281,Z 756.016,A -85,B 0,C 180,E1 -23263.342,E2 -23263.342} C_VEL
LIN {X 0,Y 164.261,Z 756.023,A -85,B 0,C 180,E1 -23266.798,E2 -23266.798} C_VEL
LIN {X 0,Y 164.29,Z 756.015,A -85,B 0,C 180,E1 -23270.355,E2 -23270.355} C_VEL
LIN {X 0,Y 164.327,Z 756.017,A -85,B 0,C 180,E1 -23274.352,E2 -23274.352} C_VEL
LIN {X 0,Y 164.358,Z 756.005,A -85,B 0,C 180,E1 -23279.128,E2 -23279.128} C_VEL
LIN {X 0,Y 164.358,Z 756.012,A -85,B 0,C 180,E1 -23284.685,E2 -23284.685} C_VEL
LIN {X 0,Y 164.419,Z 756.001,A -85,B 0,C 180,E1 -23290.117,E2 -23290.117} C_VEL
LIN {X 0,Y 164.488,Z 755.992,A -85,B 0,C 180,E1 -23295.146,E2 -23295.146} C_VEL
LIN {X 0,Y 164.766,Z 755.959,A -85,B 0,C 180,E1 -23300.176,E2 -23300.176} C_VEL
LIN {X 0,Y 164.822,Z 755.954,A -85,B 0,C 180,E1 -23302.651,E2 -23302.651} C_VEL
LIN {X 0,Y 165.276,Z 755.896,A -85,B 0,C 180,E1 -23310,E2 -23310} C_VEL
LIN {X 0,Y 164.822,Z 755.954,A -85,B 0,C 180,E1 -23317.35,E2 -23317.35} C_VEL
LIN {X 0,Y 164.704,Z 755.967,A -85,B 0,C 180,E1 -23321.06,E2 -23321.06} C_VEL
LIN {X 0,Y 164.486,Z 755.996,A -85,B 0,C 180,E1 -23327.403,E2 -23327.403} C_VEL
LIN {X 0,Y 164.476,Z 755.994,A -85,B 0,C 180,E1 -23329.989,E2 -23329.989} C_VEL
LIN {X 0,Y 164.372,Z 756.012,A -85,B 0,C 180,E1 -23336.117,E2 -23336.117} C_VEL
LIN {X 0,Y 164.393,Z 756.007,A -85,B 0,C 180,E1 -23340.776,E2 -23340.776} C_VEL
LIN {X 0,Y 168.394,Z 768.845,A -85,B 0,C 180,E1 -23343.212,E2 -23343.212} C_VEL
LIN {X 0,Y 171.561,Z 780.238,A -85,B 0,C 180,E1 -23345.715,E2 -23345.715} C_VEL
LIN {X 0,Y 173.214,Z 787.48,A -85,B 0,C 180,E1 -23347.49,E2 -23347.49} C_VEL
LIN {X 0,Y 171.199,Z 798.66,A -85,B 0,C 180,E1 -23350.239,E2 -23350.239} C_VEL
LIN {X 0,Y 169.306,Z 809.011,A -85,B 0,C 180,E1 -23353.411,E2 -23353.411} C_VEL
LIN {X 0,Y 167.523,Z 818.468,A -85,B 0,C 180,E1 -23357.021,E2 -23357.021} C_VEL
LIN {X 0,Y 166.257,Z 826.147,A -85,B 0,C 180,E1 -23360.648,E2 -23360.648} C_VEL
LIN {X 0,Y 165.478,Z 832.522,A -85,B 0,C 180,E1 -23364.421,E2 -23364.421} C_VEL
LIN {X 0,Y 165.085,Z 837.839,A -85,B 0,C 180,E1 -23368.37,E2 -23368.37} C_VEL
LIN {X 0,Y 165.362,Z 842.753,A -85,B 0,C 180,E1 -23373.192,E2 -23373.192} C_VEL
LIN {X 0,Y 166.679,Z 846.048,A -85,B 0,C 180,E1 -23378.069,E2 -23378.069} C_VEL
LIN {X 0,Y 169.042,Z 847.834,A -85,B 0,C 180,E1 -23382.989,E2 -23382.989} C_VEL
LIN {X 0,Y 170.788,Z 848.09,A -85,B 0,C 180,E1 -23385.705,E2 -23385.705} C_VEL
LIN {X 0,Y 172.772,Z 847.893,A -85,B 0,C 180,E1 -23388.264,E2 -23388.264} C_VEL
LIN {X 0,Y 177.112,Z 846.284,A -85,B 0,C 180,E1 -23392.765,E2 -23392.765} C_VEL
LIN {X 0,Y 180.384,Z 844.455,A -85,B 0,C 180,E1 -23395.531,E2 -23395.531} C_VEL
LIN {X 0,Y 185.131,Z 841.048,A -85,B 0,C 180,E1 -23398.912,E2 -23398.912} C_VEL
LIN {X 0,Y 190.371,Z 836.416,A -85,B 0,C 180,E1 -23402.115,E2 -23402.115} C_VEL
LIN {X 0,Y 196.08,Z 830.531,A -85,B 0,C 180,E1 -23405.142,E2 -23405.142} C_VEL
LIN {X 0,Y 200.178,Z 825.738,A -85,B 0,C 180,E1 -23407.058,E2 -23407.058} C_VEL
LIN {X 0,Y 201.06,Z 823.974,A -85,B 0,C 180,E1 -23408.037,E2 -23408.037} C_VEL
LIN {X 0,Y 201.734,Z 821.207,A -85,B 0,C 180,E1 -23410.031,E2 -23410.031} C_VEL
LIN {X 0,Y 202.444,Z 816.155,A -85,B 0,C 180,E1 -23414.064,E2 -23414.064} C_VEL
LIN {X 0,Y 202.113,Z 814.482,A -85,B 0,C 180,E1 -23416.151,E2 -23416.151} C_VEL
LIN {X 0,Y 200.958,Z 812.621,A -85,B 0,C 180,E1 -23420.47,E2 -23420.47} C_VEL
LIN {X 0,Y 200.021,Z 812.407,A -85,B 0,C 180,E1 -23424.938,E2 -23424.938} C_VEL
LIN {X 0,Y 199.702,Z 813.294,A -85,B 0,C 180,E1 -23428.38,E2 -23428.38} C_VEL
LIN {X 0,Y 199.639,Z 816.5,A -85,B 0,C 180,E1 -23433.068,E2 -23433.068} C_VEL
LIN {X 0,Y 199.65,Z 823.307,A -85,B 0,C 180,E1 -23438.422,E2 -23438.422} C_VEL
LIN {X 0,Y 199.544,Z 827.466,A -85,B 0,C 180,E1 -23440.845,E2 -23440.845} C_VEL
LIN {X 0,Y 199.323,Z 828.933,A -85,B 0,C 180,E1 -23441.506,E2 -23441.506} C_VEL
LIN {X 0,Y 195.397,Z 840.238,A -85,B 0,C 180,E1 -23445.464,E2 -23445.464} C_VEL
LIN {X 0,Y 191.503,Z 849.267,A -85,B 0,C 180,E1 -23448.655,E2 -23448.655} C_VEL
LIN {X 0,Y 187.226,Z 857.482,A -85,B 0,C 180,E1 -23451.731,E2 -23451.731} C_VEL
LIN {X 0,Y 182.579,Z 864.664,A -85,B 0,C 180,E1 -23454.732,E2 -23454.732} C_VEL
LIN {X 0,Y 178.201,Z 870.879,A -85,B 0,C 180,E1 -23457.83,E2 -23457.83} C_VEL
LIN {X 0,Y 174.172,Z 876.106,A -85,B 0,C 180,E1 -23461.039,E2 -23461.039} C_VEL
LIN {X 0,Y 169.251,Z 881.708,A -85,B 0,C 180,E1 -23465.465,E2 -23465.465} C_VEL
LIN {X 0,Y 167.236,Z 883.912,A -85,B 0,C 180,E1 -23467.776,E2 -23467.776} C_VEL
LIN {X 0,Y 164.657,Z 887.304,A -85,B 0,C 180,E1 -23472.615,E2 -23472.615} C_VEL
LIN {X 0,Y 163.41,Z 889.349,A -85,B 0,C 180,E1 -23477.582,E2 -23477.582} C_VEL
LIN {X 0,Y 163.526,Z 890.026,A -85,B 0,C 180,E1 -23482.592,E2 -23482.592} C_VEL
LIN {X 0,Y 164.558,Z 889.177,A -85,B 0,C 180,E1 -23487.552,E2 -23487.552} C_VEL
LIN {X 0,Y 165.284,Z 888.149,A -85,B 0,C 180,E1 -23490,E2 -23490} C_VEL
LIN {X 0,Y 164.75,Z 885.345,A -85,B 0,C 180,E1 -23493.668,E2 -23493.668} C_VEL
LIN {X 0,Y 164.313,Z 881.341,A -85,B 0,C 180,E1 -23497.372,E2 -23497.372} C_VEL
LIN {X 0,Y 164.289,Z 876.275,A -85,B 0,C 180,E1 -23500.974,E2 -23500.974} C_VEL
LIN {X 0,Y 164.873,Z 869.439,A -85,B 0,C 180,E1 -23504.818,E2 -23504.818} C_VEL
LIN {X 0,Y 166.167,Z 861.132,A -85,B 0,C 180,E1 -23508.494,E2 -23508.494} C_VEL
LIN {X 0,Y 167.019,Z 856.228,A -85,B 0,C 180,E1 -23510.313,E2 -23510.313} C_VEL
LIN {X 0,Y 167.244,Z 847.188,A -85,B 0,C 180,E1 -23513.167,E2 -23513.167} C_VEL
LIN {X 0,Y 167.313,Z 843.831,A -85,B 0,C 180,E1 -23514.099,E2 -23514.099} C_VEL
LIN {X 0,Y 166.725,Z 839.176,A -85,B 0,C 180,E1 -23515.328,E2 -23515.328} C_VEL
LIN {X 0,Y 163.888,Z 831.464,A -85,B 0,C 180,E1 -23517.256,E2 -23517.256} C_VEL
LIN {X 0,Y 160.954,Z 823.453,A -85,B 0,C 180,E1 -23519.074,E2 -23519.074} C_VEL
LIN {X 0,Y 160.227,Z 818.271,A -85,B 0,C 180,E1 -23520.095,E2 -23520.095} C_VEL
LIN {X 0,Y 160.085,Z 804.947,A -85,B 0,C 180,E1 -23522.238,E2 -23522.238} C_VEL
LIN {X 0,Y 159.704,Z 790.034,A -85,B 0,C 180,E1 -23524.015,E2 -23524.015} C_VEL
LIN {X 0,Y 159.502,Z 784.358,A -85,B 0,C 180,E1 -23524.567,E2 -23524.567} C_VEL
LIN {X 0,Y 161.388,Z 778.464,A -85,B 0,C 180,E1 -23529.289,E2 -23529.289} C_VEL
LIN {X 0,Y 161.495,Z 776.661,A -85,B 0,C 180,E1 -23530.751,E2 -23530.751} C_VEL
LIN {X 0,Y 160.215,Z 771.09,A -85,B 0,C 180,E1 -23535.424,E2 -23535.424} C_VEL
LIN {X 0,Y 159.093,Z 765.719,A -85,B 0,C 180,E1 -23540.168,E2 -23540.168} C_VEL
LIN {X 0,Y 157.893,Z 759.213,A -85,B 0,C 180,E1 -23546.194,E2 -23546.194} C_VEL
LIN {X 0,Y 157.416,Z 756.877,A -85,B 0,C 180,E1 -23548.617,E2 -23548.617} C_VEL
LIN {X 0,Y 157.316,Z 756.882,A -85,B 0,C 180,E1 -23553.465,E2 -23553.465} C_VEL
LIN {X 0,Y 157.393,Z 756.878,A -85,B 0,C 180,E1 -23559.669,E2 -23559.669} C_VEL
LIN {X 0,Y 157.455,Z 756.872,A -85,B 0,C 180,E1 -23564.466,E2 -23564.466} C_VEL
LIN {X 0,Y 157.691,Z 756.838,A -85,B 0,C 180,E1 -23569.731,E2 -23569.731} C_VEL
LIN {X 0,Y 157.768,Z 756.83,A -85,B 0,C 180,E1 -23572.32,E2 -23572.32} C_VEL
LIN {X 0,Y 158.255,Z 756.766,A -85,B 0,C 180,E1 -23580,E2 -23580} C_VEL
LIN {X 0,Y 157.762,Z 756.826,A -85,B 0,C 180,E1 -23587.681,E2 -23587.681} C_VEL
LIN {X 0,Y 157.634,Z 756.85,A -85,B 0,C 180,E1 -23591.229,E2 -23591.229} C_VEL
LIN {X 0,Y 157.434,Z 756.868,A -85,B 0,C 180,E1 -23595.536,E2 -23595.536} C_VEL
LIN {X 0,Y 157.328,Z 756.888,A -85,B 0,C 180,E1 -23600.939,E2 -23600.939} C_VEL
LIN {X 0,Y 157.267,Z 756.891,A -85,B 0,C 180,E1 -23606.649,E2 -23606.649} C_VEL
LIN {X 0,Y 157.265,Z 756.891,A -85,B 0,C 180,E1 -23612.43,E2 -23612.43} C_VEL
LIN {X 0,Y 157.259,Z 756.894,A -85,B 0,C 180,E1 -23616.445,E2 -23616.445} C_VEL
LIN {X 0,Y 157.19,Z 756.899,A -85,B 0,C 180,E1 -23622.118,E2 -23622.118} C_VEL
LIN {X 0,Y 157.19,Z 756.905,A -85,B 0,C 180,E1 -23627.883,E2 -23627.883} C_VEL
LIN {X 0,Y 157.259,Z 756.894,A -85,B 0,C 180,E1 -23633.556,E2 -23633.556} C_VEL
LIN {X 0,Y 157.276,Z 756.892,A -85,B 0,C 180,E1 -23638.107,E2 -23638.107} C_VEL
LIN {X 0,Y 157.267,Z 756.894,A -85,B 0,C 180,E1 -23643.456,E2 -23643.456} C_VEL
LIN {X 0,Y 157.361,Z 756.879,A -85,B 0,C 180,E1 -23649.702,E2 -23649.702} C_VEL
LIN {X 0,Y 157.421,Z 756.876,A -85,B 0,C 180,E1 -23654.463,E2 -23654.463} C_VEL
LIN {X 0,Y 157.689,Z 756.841,A -85,B 0,C 180,E1 -23659.731,E2 -23659.731} C_VEL
LIN {X 0,Y 157.76,Z 756.833,A -85,B 0,C 180,E1 -23662.32,E2 -23662.32} C_VEL
LIN {X 0,Y 158.238,Z 756.773,A -85,B 0,C 180,E1 -23670,E2 -23670} C_VEL
LIN {X 0,Y 157.761,Z 756.834,A -85,B 0,C 180,E1 -23677.681,E2 -23677.681} C_VEL
LIN {X 0,Y 157.639,Z 756.847,A -85,B 0,C 180,E1 -23681.236,E2 -23681.236} C_VEL
LIN {X 0,Y 157.445,Z 756.872,A -85,B 0,C 180,E1 -23685.535,E2 -23685.535} C_VEL
LIN {X 0,Y 157.37,Z 756.878,A -85,B 0,C 180,E1 -23690.933,E2 -23690.933} C_VEL
LIN {X 0,Y 157.312,Z 756.889,A -85,B 0,C 180,E1 -23696.681,E2 -23696.681} C_VEL
LIN {X 0,Y 157.342,Z 756.886,A -85,B 0,C 180,E1 -23699.981,E2 -23699.981} C_VEL
LIN {X 0,Y 161.171,Z 769.156,A -85,B 0,C 180,E1 -23702.405,E2 -23702.405} C_VEL
LIN {X 0,Y 164.433,Z 780.744,A -85,B 0,C 180,E1 -23705.053,E2 -23705.053} C_VEL
LIN {X 0,Y 166.052,Z 787.453,A -85,B 0,C 180,E1 -23706.755,E2 -23706.755} C_VEL
LIN {X 0,Y 166.184,Z 788.93,A -85,B 0,C 180,E1 -23707.141,E2 -23707.141} C_VEL
LIN {X 0,Y 163.986,Z 800.558,A -85,B 0,C 180,E1 -23710.139,E2 -23710.139} C_VEL
LIN {X 0,Y 162.067,Z 810.708,A -85,B 0,C 180,E1 -23713.444,E2 -23713.444} C_VEL
LIN {X 0,Y 160.323,Z 819.771,A -85,B 0,C 180,E1 -23717.103,E2 -23717.103} C_VEL
LIN {X 0,Y 159.062,Z 827.525,A -85,B 0,C 180,E1 -23720.977,E2 -23720.977} C_VEL
LIN {X 0,Y 158.247,Z 834.683,A -85,B 0,C 180,E1 -23725.511,E2 -23725.511} C_VEL
LIN {X 0,Y 157.985,Z 839.354,A -85,B 0,C 180,E1 -23729.23,E2 -23729.23} C_VEL
LIN {X 0,Y 158.36,Z 843.664,A -85,B 0,C 180,E1 -23733.653,E2 -23733.653} C_VEL
LIN {X 0,Y 159.46,Z 846.539,A -85,B 0,C 180,E1 -23737.753,E2 -23737.753} C_VEL
LIN {X 0,Y 161.81,Z 848.707,A -85,B 0,C 180,E1 -23742.852,E2 -23742.852} C_VEL
LIN {X 0,Y 165.286,Z 849.315,A -85,B 0,C 180,E1 -23747.952,E2 -23747.952} C_VEL
LIN {X 0,Y 167.365,Z 848.99,A -85,B 0,C 180,E1 -23750.33,E2 -23750.33} C_VEL
LIN {X 0,Y 169.962,Z 848.169,A -85,B 0,C 180,E1 -23752.94,E2 -23752.94} C_VEL
LIN {X 0,Y 172.722,Z 846.964,A -85,B 0,C 180,E1 -23755.332,E2 -23755.332} C_VEL
LIN {X 0,Y 177.473,Z 844.156,A -85,B 0,C 180,E1 -23758.865,E2 -23758.865} C_VEL
LIN {X 0,Y 182.865,Z 840.185,A -85,B 0,C 180,E1 -23762.202,E2 -23762.202} C_VEL
LIN {X 0,Y 188.707,Z 834.969,A -85,B 0,C 180,E1 -23765.342,E2 -23765.342} C_VEL
LIN {X 0,Y 194.979,Z 828.374,A -85,B 0,C 180,E1 -23768.29,E2 -23768.29} C_VEL
LIN {X 0,Y 195.767,Z 826.87,A -85,B 0,C 180,E1 -23769.297,E2 -23769.297} C_VEL
LIN {X 0,Y 197.032,Z 822.323,A -85,B 0,C 180,E1 -23773.164,E2 -23773.164} C_VEL
LIN {X 0,Y 197.375,Z 820.939,A -85,B 0,C 180,E1 -23774.433,E2 -23774.433} C_VEL
LIN {X 0,Y 197.147,Z 819.467,A -85,B 0,C 180,E1 -23776.57,E2 -23776.57} C_VEL
LIN {X 0,Y 196.749,Z 818.58,A -85,B 0,C 180,E1 -23778.753,E2 -23778.753} C_VEL
LIN {X 0,Y 196.192,Z 817.971,A -85,B 0,C 180,E1 -23781.348,E2 -23781.348} C_VEL
LIN {X 0,Y 195.57,Z 818.149,A -85,B 0,C 180,E1 -23785.546,E2 -23785.546} C_VEL
LIN {X 0,Y 195.391,Z 818.766,A -85,B 0,C 180,E1 -23787.878,E2 -23787.878} C_VEL
LIN {X 0,Y 195.214,Z 820.112,A -85,B 0,C 180,E1 -23790.266,E2 -23790.266} C_VEL
LIN {X 0,Y 195.17,Z 821.896,A -85,B 0,C 180,E1 -23792.693,E2 -23792.693} C_VEL
LIN {X 0,Y 194.817,Z 828.097,A -85,B 0,C 180,E1 -23797.826,E2 -23797.826} C_VEL
LIN {X 0,Y 194.505,Z 831.441,A -85,B 0,C 180,E1 -23799.923,E2 -23799.923} C_VEL
LIN {X 0,Y 194.127,Z 833.046,A -85,B 0,C 180,E1 -23800.667,E2 -23800.667} C_VEL
LIN {X 0,Y 189.669,Z 843.465,A -85,B 0,C 180,E1 -23804.573,E2 -23804.573} C_VEL
LIN {X 0,Y 185.497,Z 851.766,A -85,B 0,C 180,E1 -23807.739,E2 -23807.739} C_VEL
LIN {X 0,Y 179.653,Z 861.242,A -85,B 0,C 180,E1 -23811.677,E2 -23811.677} C_VEL
LIN {X 0,Y 173.619,Z 869.046,A -85,B 0,C 180,E1 -23815.478,E2 -23815.478} C_VEL
LIN {X 0,Y 169.377,Z 874.34,A -85,B 0,C 180,E1 -23818.757,E2 -23818.757} C_VEL
LIN {X 0,Y 163.955,Z 880.013,A -85,B 0,C 180,E1 -23823.25,E2 -23823.25} C_VEL
LIN {X 0,Y 160.653,Z 883.256,A -85,B 0,C 180,E1 -23826.813,E2 -23826.813} C_VEL
LIN {X 0,Y 157.848,Z 886.451,A -85,B 0,C 180,E1 -23831.84,E2 -23831.84} C_VEL
LIN {X 0,Y 156.453,Z 888.274,A -85,B 0,C 180,E1 -23837.02,E2 -23837.02} C_VEL
LIN {X 0,Y 156.501,Z 888.717,A -85,B 0,C 180,E1 -23842.257,E2 -23842.257} C_VEL
LIN {X 0,Y 157.572,Z 887.733,A -85,B 0,C 180,E1 -23847.443,E2 -23847.443} C_VEL
LIN {X 0,Y 158.311,Z 886.65,A -85,B 0,C 180,E1 -23850,E2 -23850} C_VEL
LIN {X 0,Y 157.77,Z 883.67,A -85,B 0,C 180,E1 -23853.831,E2 -23853.831} C_VEL
LIN {X 0,Y 157.3,Z 879.464,A -85,B 0,C 180,E1 -23857.703,E2 -23857.703} C_VEL
LIN {X 0,Y 157.388,Z 873.012,A -85,B 0,C 180,E1 -23862.18,E2 -23862.18} C_VEL
LIN {X 0,Y 158.227,Z 865.744,A -85,B 0,C 180,E1 -23866.117,E2 -23866.117} C_VEL
LIN {X 0,Y 159.509,Z 858.473,A -85,B 0,C 180,E1 -23869.296,E2 -23869.296} C_VEL
LIN {X 0,Y 160.057,Z 853.292,A -85,B 0,C 180,E1 -23871.219,E2 -23871.219} C_VEL
LIN {X 0,Y 160.291,Z 842.357,A -85,B 0,C 180,E1 -23874.616,E2 -23874.616} C_VEL
LIN {X 0,Y 160.29,Z 831.399,A -85,B 0,C 180,E1 -23877.411,E2 -23877.411} C_VEL
LIN {X 0,Y 160.24,Z 819.184,A -85,B 0,C 180,E1 -23879.927,E2 -23879.927} C_VEL
LIN {X 0,Y 160.227,Z 818.271,A -85,B 0,C 180,E1 -23880.095,E2 -23880.095} C_VEL
LIN {X 0,Y 159.491,Z 813.056,A -85,B 0,C 180,E1 -23881.062,E2 -23881.062} C_VEL
LIN {X 0,Y 156.516,Z 804.602,A -85,B 0,C 180,E1 -23882.62,E2 -23882.62} C_VEL
LIN {X 0,Y 153.596,Z 795.922,A -85,B 0,C 180,E1 -23884.029,E2 -23884.029} C_VEL
LIN {X 0,Y 152.882,Z 790.357,A -85,B 0,C 180,E1 -23884.718,E2 -23884.718} C_VEL
LIN {X 0,Y 152.666,Z 783.378,A -85,B 0,C 180,E1 -23885.436,E2 -23885.436} C_VEL
LIN {X 0,Y 154.332,Z 778.402,A -85,B 0,C 180,E1 -23889.608,E2 -23889.608} C_VEL
LIN {X 0,Y 154.066,Z 775.479,A -85,B 0,C 180,E1 -23892.134,E2 -23892.134} C_VEL
LIN {X 0,Y 152.395,Z 768.304,A -85,B 0,C 180,E1 -23898.576,E2 -23898.576} C_VEL
LIN {X 0,Y 151.191,Z 762.115,A -85,B 0,C 180,E1 -23904.475,E2 -23904.475} C_VEL
LIN {X 0,Y 150.356,Z 757.757,A -85,B 0,C 180,E1 -23909.059,E2 -23909.059} C_VEL
LIN {X 0,Y 150.219,Z 757.77,A -85,B 0,C 180,E1 -23915.098,E2 -23915.098} C_VEL
LIN {X 0,Y 150.36,Z 757.749,A -85,B 0,C 180,E1 -23920.902,E2 -23920.902} C_VEL
LIN {X 0,Y 150.437,Z 757.746,A -85,B 0,C 180,E1 -23926.492,E2 -23926.492} C_VEL
LIN {X 0,Y 150.613,Z 757.719,A -85,B 0,C 180,E1 -23929.243,E2 -23929.243} C_VEL
LIN {X 0,Y 150.705,Z 757.708,A -85,B 0,C 180,E1 -23931.958,E2 -23931.958} C_VEL
LIN {X 0,Y 151.216,Z 757.643,A -85,B 0,C 180,E1 -23940,E2 -23940} C_VEL
LIN {X 0,Y 150.7,Z 757.706,A -85,B 0,C 180,E1 -23948.043,E2 -23948.043} C_VEL
LIN {X 0,Y 150.575,Z 757.728,A -85,B 0,C 180,E1 -23951.432,E2 -23951.432} C_VEL
LIN {X 0,Y 150.344,Z 757.75,A -85,B 0,C 180,E1 -23956.289,E2 -23956.289} C_VEL
LIN {X 0,Y 150.299,Z 757.763,A -85,B 0,C 180,E1 -23960.739,E2 -23960.739} C_VEL
LIN {X 0,Y 150.185,Z 757.775,A -85,B 0,C 180,E1 -23967.237,E2 -23967.237} C_VEL
LIN {X 0,Y 150.206,Z 757.77,A -85,B 0,C 180,E1 -23972.626,E2 -23972.626} C_VEL
LIN {X 0,Y 150.169,Z 757.779,A -85,B 0,C 180,E1 -23977.475,E2 -23977.475} C_VEL
LIN {X 0,Y 150.133,Z 757.78,A -85,B 0,C 180,E1 -23981.497,E2 -23981.497} C_VEL
LIN {X 0,Y 150.127,Z 757.783,A -85,B 0,C 180,E1 -23985.396,E2 -23985.396} C_VEL
LIN {X 0,Y 150.137,Z 757.78,A -85,B 0,C 180,E1 -23989.054,E2 -23989.054} C_VEL
LIN {X 0,Y 150.176,Z 757.776,A -85,B 0,C 180,E1 -23992.71,E2 -23992.71} C_VEL
LIN {X 0,Y 150.203,Z 757.773,A -85,B 0,C 180,E1 -23997.376,E2 -23997.376} C_VEL
LIN {X 0,Y 150.183,Z 757.777,A -85,B 0,C 180,E1 -24002.765,E2 -24002.765} C_VEL
LIN {X 0,Y 150.284,Z 757.761,A -85,B 0,C 180,E1 -24009.277,E2 -24009.277} C_VEL
LIN {X 0,Y 150.325,Z 757.758,A -85,B 0,C 180,E1 -24013.709,E2 -24013.709} C_VEL
LIN {X 0,Y 150.61,Z 757.724,A -85,B 0,C 180,E1 -24019.243,E2 -24019.243} C_VEL
LIN {X 0,Y 150.683,Z 757.714,A -85,B 0,C 180,E1 -24021.957,E2 -24021.957} C_VEL
LIN {X 0,Y 151.199,Z 757.65,A -85,B 0,C 180,E1 -24030,E2 -24030} C_VEL
LIN {X 0,Y 150.684,Z 757.714,A -85,B 0,C 180,E1 -24038.044,E2 -24038.044} C_VEL
LIN {X 0,Y 150.579,Z 757.725,A -85,B 0,C 180,E1 -24041.436,E2 -24041.436} C_VEL
LIN {X 0,Y 150.356,Z 757.755,A -85,B 0,C 180,E1 -24046.288,E2 -24046.288} C_VEL
LIN {X 0,Y 150.352,Z 757.752,A -85,B 0,C 180,E1 -24050.791,E2 -24050.791} C_VEL
LIN {X 0,Y 150.242,Z 757.77,A -85,B 0,C 180,E1 -24057.279,E2 -24057.279} C_VEL
LIN {X 0,Y 150.291,Z 757.941,A -85,B 0,C 180,E1 -24059.215,E2 -24059.215} C_VEL
LIN {X 0,Y 154.04,Z 769.775,A -85,B 0,C 180,E1 -24061.647,E2 -24061.647} C_VEL
LIN {X 0,Y 157.272,Z 781.124,A -85,B 0,C 180,E1 -24064.345,E2 -24064.345} C_VEL
LIN {X 0,Y 159.226,Z 789.511,A -85,B 0,C 180,E1 -24066.567,E2 -24066.567} C_VEL
LIN {X 0,Y 157.163,Z 800.221,A -85,B 0,C 180,E1 -24069.421,E2 -24069.421} C_VEL
LIN {X 0,Y 155.227,Z 810.407,A -85,B 0,C 180,E1 -24072.777,E2 -24072.777} C_VEL
LIN {X 0,Y 153.378,Z 819.674,A -85,B 0,C 180,E1 -24076.581,E2 -24076.581} C_VEL
LIN {X 0,Y 151.942,Z 828.225,A -85,B 0,C 180,E1 -24080.945,E2 -24080.945} C_VEL
LIN {X 0,Y 151.202,Z 834.949,A -85,B 0,C 180,E1 -24085.292,E2 -24085.292} C_VEL
LIN {X 0,Y 150.898,Z 839.771,A -85,B 0,C 180,E1 -24089.181,E2 -24089.181} C_VEL
LIN {X 0,Y 151.323,Z 844.251,A -85,B 0,C 180,E1 -24093.818,E2 -24093.818} C_VEL
LIN {X 0,Y 152.575,Z 847.475,A -85,B 0,C 180,E1 -24098.376,E2 -24098.376} C_VEL
LIN {X 0,Y 154.573,Z 849.491,A -85,B 0,C 180,E1 -24102.712,E2 -24102.712} C_VEL
LIN {X 0,Y 158.076,Z 850.536,A -85,B 0,C 180,E1 -24107.993,E2 -24107.993} C_VEL
LIN {X 0,Y 162.183,Z 850.07,A -85,B 0,C 180,E1 -24112.53,E2 -24112.53} C_VEL
LIN {X 0,Y 165.019,Z 849.196,A -85,B 0,C 180,E1 -24115.113,E2 -24115.113} C_VEL
LIN {X 0,Y 168.771,Z 847.517,A -85,B 0,C 180,E1 -24118.055,E2 -24118.055} C_VEL
LIN {X 0,Y 173.417,Z 844.86,A -85,B 0,C 180,E1 -24121.161,E2 -24121.161} C_VEL
LIN {X 0,Y 179.237,Z 840.712,A -85,B 0,C 180,E1 -24124.498,E2 -24124.498} C_VEL
LIN {X 0,Y 184.982,Z 835.855,A -85,B 0,C 180,E1 -24127.361,E2 -24127.361} C_VEL
LIN {X 0,Y 188.93,Z 832.119,A -85,B 0,C 180,E1 -24129.096,E2 -24129.096} C_VEL
LIN {X 0,Y 189.804,Z 831.11,A -85,B 0,C 180,E1 -24129.591,E2 -24129.591} C_VEL
LIN {X 0,Y 190.91,Z 828.706,A -85,B 0,C 180,E1 -24131.681,E2 -24131.681} C_VEL
LIN {X 0,Y 192.126,Z 825.539,A -85,B 0,C 180,E1 -24134.836,E2 -24134.836} C_VEL
LIN {X 0,Y 191.917,Z 824.037,A -85,B 0,C 180,E1 -24137.8,E2 -24137.8} C_VEL
LIN {X 0,Y 191.392,Z 823.222,A -85,B 0,C 180,E1 -24141.543,E2 -24141.543} C_VEL
LIN {X 0,Y 191.035,Z 823.277,A -85,B 0,C 180,E1 -24143.871,E2 -24143.871} C_VEL
LIN {X 0,Y 190.771,Z 824.209,A -85,B 0,C 180,E1 -24147.851,E2 -24147.851} C_VEL
LIN {X 0,Y 190.457,Z 826.749,A -85,B 0,C 180,E1 -24151.927,E2 -24151.927} C_VEL
LIN {X 0,Y 189.771,Z 831.617,A -85,B 0,C 180,E1 -24156.338,E2 -24156.338} C_VEL
LIN {X 0,Y 189.41,Z 835.058,A -85,B 0,C 180,E1 -24158.812,E2 -24158.812} C_VEL
LIN {X 0,Y 189.1,Z 836.3,A -85,B 0,C 180,E1 -24159.527,E2 -24159.527} C_VEL
LIN {X 0,Y 184.104,Z 846.2,A -85,B 0,C 180,E1 -24163.505,E2 -24163.505} C_VEL
LIN {X 0,Y 179.486,Z 854.039,A -85,B 0,C 180,E1 -24166.745,E2 -24166.745} C_VEL
LIN {X 0,Y 173.874,Z 862.071,A -85,B 0,C 180,E1 -24170.37,E2 -24170.37} C_VEL
LIN {X 0,Y 167.79,Z 869.203,A -85,B 0,C 180,E1 -24174.098,E2 -24174.098} C_VEL
LIN {X 0,Y 161.832,Z 875.666,A -85,B 0,C 180,E1 -24178.591,E2 -24178.591} C_VEL
LIN {X 0,Y 156.384,Z 880.672,A -85,B 0,C 180,E1 -24183.294,E2 -24183.294} C_VEL
LIN {X 0,Y 154.136,Z 882.631,A -85,B 0,C 180,E1 -24185.772,E2 -24185.772} C_VEL
LIN {X 0,Y 151.072,Z 885.533,A -85,B 0,C 180,E1 -24190.995,E2 -24190.995} C_VEL
LIN {X 0,Y 149.522,Z 887.128,A -85,B 0,C 180,E1 -24196.407,E2 -24196.407} C_VEL
LIN {X 0,Y 149.469,Z 887.414,A -85,B 0,C 180,E1 -24201.891,E2 -24201.891} C_VEL
LIN {X 0,Y 150.576,Z 886.244,A -85,B 0,C 180,E1 -24207.324,E2 -24207.324} C_VEL
LIN {X 0,Y 151.337,Z 885.023,A -85,B 0,C 180,E1 -24210,E2 -24210} C_VEL
LIN {X 0,Y 150.782,Z 881.886,A -85,B 0,C 180,E1 -24214.009,E2 -24214.009} C_VEL
LIN {X 0,Y 150.307,Z 877.48,A -85,B 0,C 180,E1 -24218.063,E2 -24218.063} C_VEL
LIN {X 0,Y 150.514,Z 870.724,A -85,B 0,C 180,E1 -24222.813,E2 -24222.813} C_VEL
LIN {X 0,Y 151.475,Z 863.307,A -85,B 0,C 180,E1 -24226.857,E2 -24226.857} C_VEL
LIN {X 0,Y 152.765,Z 855.701,A -85,B 0,C 180,E1 -24230.184,E2 -24230.184} C_VEL
LIN {X 0,Y 153.079,Z 847.655,A -85,B 0,C 180,E1 -24233.084,E2 -24233.084} C_VEL
LIN {X 0,Y 153.19,Z 837.253,A -85,B 0,C 180,E1 -24236.204,E2 -24236.204} C_VEL
LIN {X 0,Y 153.332,Z 825.292,A -85,B 0,C 180,E1 -24239.147,E2 -24239.147} C_VEL
LIN {X 0,Y 153.206,Z 812.494,A -85,B 0,C 180,E1 -24241.646,E2 -24241.646} C_VEL
LIN {X 0,Y 153.096,Z 799.287,A -85,B 0,C 180,E1 -24243.662,E2 -24243.662} C_VEL
LIN {X 0,Y 152.882,Z 790.357,A -85,B 0,C 180,E1 -24244.718,E2 -24244.718} C_VEL
LIN {X 0,Y 152.564,Z 786.947,A -85,B 0,C 180,E1 -24245.319,E2 -24245.319} C_VEL
LIN {X 0,Y 151.598,Z 783.441,A -85,B 0,C 180,E1 -24246.495,E2 -24246.495} C_VEL
LIN {X 0,Y 150.329,Z 780.688,A -85,B 0,C 180,E1 -24247.96,E2 -24247.96} C_VEL
LIN {X 0,Y 146.83,Z 774.934,A -85,B 0,C 180,E1 -24253.065,E2 -24253.065} C_VEL
LIN {X 0,Y 146.278,Z 773.253,A -85,B 0,C 180,E1 -24254.614,E2 -24254.614} C_VEL
LIN {X 0,Y 144.864,Z 766.69,A -85,B 0,C 180,E1 -24260.917,E2 -24260.917} C_VEL
LIN {X 0,Y 143.897,Z 761.547,A -85,B 0,C 180,E1 -24266.128,E2 -24266.128} C_VEL
LIN {X 0,Y 143.271,Z 758.639,A -85,B 0,C 180,E1 -24269.407,E2 -24269.407} C_VEL
LIN {X 0,Y 143.157,Z 758.647,A -85,B 0,C 180,E1 -24273.779,E2 -24273.779} C_VEL
LIN {X 0,Y 143.307,Z 758.632,A -85,B 0,C 180,E1 -24279.923,E2 -24279.923} C_VEL
LIN {X 0,Y 143.36,Z 758.627,A -85,B 0,C 180,E1 -24285.811,E2 -24285.811} C_VEL
LIN {X 0,Y 143.539,Z 758.601,A -85,B 0,C 180,E1 -24288.706,E2 -24288.706} C_VEL
LIN {X 0,Y 143.627,Z 758.589,A -85,B 0,C 180,E1 -24291.559,E2 -24291.559} C_VEL
LIN {X 0,Y 144.174,Z 758.52,A -85,B 0,C 180,E1 -24300,E2 -24300} C_VEL
LIN {X 0,Y 143.622,Z 758.588,A -85,B 0,C 180,E1 -24308.442,E2 -24308.442} C_VEL
LIN {X 0,Y 143.502,Z 758.609,A -85,B 0,C 180,E1 -24311.622,E2 -24311.622} C_VEL
LIN {X 0,Y 143.281,Z 758.632,A -85,B 0,C 180,E1 -24317.116,E2 -24317.116} C_VEL
LIN {X 0,Y 143.236,Z 758.644,A -85,B 0,C 180,E1 -24321.212,E2 -24321.212} C_VEL
LIN {X 0,Y 143.142,Z 758.654,A -85,B 0,C 180,E1 -24327.9,E2 -24327.9} C_VEL
LIN {X 0,Y 143.136,Z 758.65,A -85,B 0,C 180,E1 -24333.415,E2 -24333.415} C_VEL
LIN {X 0,Y 143.052,Z 758.665,A -85,B 0,C 180,E1 -24339.694,E2 -24339.694} C_VEL
LIN {X 0,Y 143.034,Z 758.663,A -85,B 0,C 180,E1 -24343.464,E2 -24343.464} C_VEL
LIN {X 0,Y 143.038,Z 758.667,A -85,B 0,C 180,E1 -24347.478,E2 -24347.478} C_VEL
LIN {X 0,Y 143.072,Z 758.657,A -85,B 0,C 180,E1 -24351.81,E2 -24351.81} C_VEL
LIN {X 0,Y 143.171,Z 758.649,A -85,B 0,C 180,E1 -24357.319,E2 -24357.319} C_VEL
LIN {X 0,Y 143.106,Z 758.658,A -85,B 0,C 180,E1 -24363.769,E2 -24363.769} C_VEL
LIN {X 0,Y 143.249,Z 758.637,A -85,B 0,C 180,E1 -24369.914,E2 -24369.914} C_VEL
LIN {X 0,Y 143.316,Z 758.628,A -85,B 0,C 180,E1 -24375.807,E2 -24375.807} C_VEL
LIN {X 0,Y 143.536,Z 758.602,A -85,B 0,C 180,E1 -24378.706,E2 -24378.706} C_VEL
LIN {X 0,Y 143.609,Z 758.596,A -85,B 0,C 180,E1 -24381.558,E2 -24381.558} C_VEL
LIN {X 0,Y 144.157,Z 758.527,A -85,B 0,C 180,E1 -24390,E2 -24390} C_VEL
LIN {X 0,Y 143.61,Z 758.595,A -85,B 0,C 180,E1 -24398.443,E2 -24398.443} C_VEL
LIN {X 0,Y 143.506,Z 758.605,A -85,B 0,C 180,E1 -24401.627,E2 -24401.627} C_VEL
LIN {X 0,Y 143.298,Z 758.634,A -85,B 0,C 180,E1 -24407.114,E2 -24407.114} C_VEL
LIN {X 0,Y 143.277,Z 758.634,A -85,B 0,C 180,E1 -24411.252,E2 -24411.252} C_VEL
LIN {X 0,Y 143.209,Z 758.776,A -85,B 0,C 180,E1 -24418.314,E2 -24418.314} C_VEL
LIN {X 0,Y 147.075,Z 770.766,A -85,B 0,C 180,E1 -24420.911,E2 -24420.911} C_VEL
LIN {X 0,Y 150.214,Z 782.141,A -85,B 0,C 180,E1 -24423.752,E2 -24423.752} C_VEL
LIN {X 0,Y 152.228,Z 790.407,A -85,B 0,C 180,E1 -24426.061,E2 -24426.061} C_VEL
LIN {X 0,Y 149.961,Z 802.139,A -85,B 0,C 180,E1 -24429.35,E2 -24429.35} C_VEL
LIN {X 0,Y 147.856,Z 812.613,A -85,B 0,C 180,E1 -24433.044,E2 -24433.044} C_VEL
LIN {X 0,Y 146.131,Z 821.254,A -85,B 0,C 180,E1 -24436.817,E2 -24436.817} C_VEL
LIN {X 0,Y 144.842,Z 828.877,A -85,B 0,C 180,E1 -24440.928,E2 -24440.928} C_VEL
LIN {X 0,Y 144.112,Z 835.397,A -85,B 0,C 180,E1 -24445.265,E2 -24445.265} C_VEL
